// TwinCAT 3 PLC project _710_Clamping
// ProgramVersion: 3.1.4024.0
// libraries:
//   Tc2_Standard, * (Beckhoff Automation GmbH)
//   Tc2_System, * (Beckhoff Automation GmbH)
//   Tc3_Module, * (Beckhoff Automation GmbH)
//   VisuDialogs, * (System)
// project tree:
//   DUTs/ udt_MH_Robot_Input.TcDUT (not stored), udt_HDL_PartData.TcDUT, udt_MH_Robot_Output.TcDUT (not stored)
//   / GlobalTextList.TcGTLO, PlcTask.TcTTO, Visualization Manager.TcVMO (not stored)
//   GVLs/ Inputs.TcGVL (not stored), Memory_DB.TcGVL (not stored), Outputs.TcGVL (not stored)
//   POUs/ Fixture1_Auto.TcPOU, Callblocks.TcPOU, Callblocks_FX1.TcPOU, Callblocks_FX2.TcPOU, Clamp.TcPOU (not stored), Feedback_FB.TcPOU (not stored), Fixture2_Auto.TcPOU (not stored), FX2TextList.TcTLO, MAIN.TcPOU (not stored), MHRobot.TcPOU (not stored), Mode.TcPOU, RollerDoor.TcPOU, FX1TextList.TcTLO, Trunion.TcPOU, Turntable.TcPOU (not stored), WeldRobot.TcPOU (not stored)
//   VISUs/ Fixture_Auto.TcVIS, Fixture_Manual.TcVIS
// real-time tasks:
//   TASK PlcTask: cycle T#10ms, priority 20, ADS port 350

CONFIGURATION _710_Clamping
    RESOURCE PLC ON TwinCAT3
        TASK PlcTask(INTERVAL := T#10ms, PRIORITY := 20);
        PROGRAM MAIN WITH PlcTask : MAIN;
    END_RESOURCE
END_CONFIGURATION

// ---- DUTs/udt_HDL_PartData.TcDUT
TYPE udt_HDL_PartData :
STRUCT
	
PartId	:DINT;
State	:BOOL;
Varient	:BOOL;
Exists	:BOOL;

	
END_STRUCT
END_TYPE

// ---- POUs/Fixture1_Auto.TcPOU
PROGRAM Fixture1_Auto
VAR
	
nState_Door    : INT; // 0: Idle, 10: Starting, 20: Rotating, 30: Stopping
	
END_VAR




/////////////// OPERATOR LOAD PART FIX 1 ///////////////

		IF Memory_DB.M_Auto_Active AND 
		   Memory_DB.M_Power_On AND 
		   Inputs.i_Front_Door_Up
		   THEN   
		IF Memory_DB.M_FX1_LOAD1 AND Memory_DB.M_Turntable_POS1_Reached AND Memory_DB.M_Fixture1_TR_POS1_Reached  THEN
		  Inputs.i_FX1_PART_CONTROL_B1 := TRUE;
		  Inputs.i_FX1_PART_CONTROL_B2 := TRUE;
		  Inputs.i_FX1_PART_CONTROL_B3 := TRUE;
		  Inputs.i_FX1_PART_CONTROL_B4 := TRUE;
		  Inputs.i_FX1_PART_CONTROL_B5 := TRUE;
		  Inputs.i_FX1_PART_CONTROL_B6 := TRUE;
		  Inputs.i_FX1_PART_CONTROL_B7 := TRUE;
		  Memory_DB.M_FX1_LOAD1_COMPLETED :=TRUE;
		
		ELSIF Memory_DB.M_Auto_Active AND Memory_DB.M_Turntable_POS1_Reached AND Memory_DB.M_Fixture1_TR_POS2_Reached AND Memory_DB.M_FX1_LOAD2 THEN
		      Inputs.i_FX1_PART_CONTROL_B15 := TRUE;
		      Inputs.i_FX1_PART_CONTROL_B16 := TRUE;
		      Inputs.i_FX1_PART_CONTROL_B17 := TRUE;
		      Inputs.i_FX1_PART_CONTROL_B18 := TRUE;
		      Inputs.i_FX1_PART_CONTROL_B19 := TRUE;
		      Inputs.i_FX1_PART_CONTROL_B20 := TRUE;
		      Inputs.i_FX1_PART_CONTROL_B21 := TRUE;
		      Memory_DB.M_FX1_LOAD2_COMPLETED :=TRUE;
		
		ELSIF Memory_DB.M_FX1_LOAD1_COMPLETED AND Memory_DB.M_FX1_LOAD2_COMPLETED THEN
			
			  Memory_DB.M_Fixture1_TR_Start :=TRUE;
			
		END_IF;
		END_IF;
		 IF 
		   Memory_DB. M_FX1_All_Initialise THEN
		   Memory_DB.M_Turntable_Start := TRUE;
	       Memory_DB.M_Turntable_POS1_CMD := TRUE;
		   Memory_DB.M_Turntable_POS2_CMD := FALSE;
		   Memory_DB.M_Fixture1_TR_Start := TRUE;
	       Memory_DB.M_Fixture1_TR_POS1_CMD := TRUE;
		   Memory_DB.M_Fixture1_TR_POS2_CMD := FALSE;
		   Memory_DB.M_REAR_DOOR_DOWN := TRUE;
		   Memory_DB.M_REAR_DOOR_Up := FALSE;
		   
		 END_IF
//////////////////LODING SIDE DOOR & TRUNION CONTROL OPERATION/////////////////
IF  Memory_DB.M_Auto_Active AND Memory_DB.M_Safety_Ok AND Memory_DB.M_Power_On  THEN
	
CASE nState_Door  OF
    0: // Default Position1 of Door Open
	IF Memory_DB.M_Turntable_POS1_Reached AND Memory_DB.M_Fixture1_TR_POS1_Reached THEN      
		Memory_DB.M_FRONT_DOOR_Down	:=FALSE;
		Memory_DB.M_FRONT_DOOR_UP	:=TRUE;	
		Memory_DB.M_R03_MH_Goto_Drop2:=FALSE;
		nState_Door := 10;
     END_IF  
	 
    10: // 1st Load completed and Door Close Command
 
        IF Memory_DB.M_FX1_LOAD1_COMPLETED AND Memory_DB.M_FX1_Cycle_Start_PB AND Inputs.i_Front_Door_Up THEN
		Memory_DB.M_FRONT_DOOR_Down	:=TRUE;
		Memory_DB.M_FRONT_DOOR_UP	:=FALSE;

            nState_Door := 20; // Trunion Move
        END_IF
		       
    20: // Clamp Sequence at Trunion Pos1
 
        IF Inputs.i_Front_Door_Down AND Memory_DB.M_Fixture1_TR_POS1_Reached THEN
		Memory_DB.A_FX1_CC1_CLAMPING_UNIT1_3_WP:=TRUE;
		Memory_DB.A_FX1_CC3_CLAMPING_UNIT3_3_WP:=TRUE;
		Memory_DB.A_FX1_CC5_CLAMPING_UNIT5_1_WP:=TRUE;
		Memory_DB.A_FX1_CC1_CLAMPING_UNIT1_3_HP:=FALSE;
		Memory_DB.A_FX1_CC3_CLAMPING_UNIT3_3_HP:=FALSE;
		Memory_DB.A_FX1_CC5_CLAMPING_UNIT5_1_HP:=FALSE;		

         nState_Door := 30; // Error State
        END_IF	

        
    30: // Trunion move to Position 2 for 2nd Load
 
        IF Inputs.i_Front_Door_Down AND Inputs.i_FX1_CC1_Clamp_1_Sensor_WP AND 
		Inputs.i_FX1_CC3_Clamp_1_Sensor_WP AND Inputs.i_FX1_CC5_Clamp_1_Sensor_WP THEN
		Memory_DB.M_Fixture1_TR_POS2_CMD:=TRUE;
		Memory_DB.M_Fixture1_TR_POS1_CMD:=FALSE;

            nState_Door := 40; // Error State
        END_IF		
        
    40: // Door Open command for 2nd Load
 
        IF Memory_DB.M_Fixture1_TR_POS2_Reached AND Inputs.i_Front_Door_Down THEN
		Memory_DB.M_FRONT_DOOR_Down:=FALSE;
		Memory_DB.M_FRONT_DOOR_UP  :=TRUE;

            nState_Door := 50; // Error State
        END_IF	
        
    50: // 2nd Load completed on Trunion & Door Close Command
 
        IF Memory_DB.M_FX1_LOAD2_COMPLETED AND Memory_DB.M_FX1_Cycle_Start_PB AND Inputs.i_Front_Door_Up THEN
		Memory_DB.M_FRONT_DOOR_Down      :=TRUE;
		Memory_DB.M_FRONT_DOOR_Up        :=FALSE;

            nState_Door := 60; // Error State
        END_IF
		
    60: // Clamp Sequence at Trunion Pos1
 
        IF Inputs.i_Front_Door_Down AND Memory_DB.M_Fixture1_TR_POS2_Reached THEN
		Memory_DB.A_FX1_CC2_CLAMPING_UNIT2_3_WP:=TRUE;
		Memory_DB.A_FX1_CC4_CLAMPING_UNIT4_3_WP:=TRUE;
		Memory_DB.A_FX1_CC6_CLAMPING_UNIT6_1_WP:=TRUE;
		Memory_DB.A_FX1_CC2_CLAMPING_UNIT2_3_HP:=FALSE;
		Memory_DB.A_FX1_CC4_CLAMPING_UNIT4_3_HP:=FALSE;
		Memory_DB.A_FX1_CC6_CLAMPING_UNIT6_1_HP:=FALSE;	

         nState_Door := 70; // Error State
        END_IF		
        
    70: // Move Trunion to Default/Pos1
 
        IF Memory_DB.M_Fixture1_TR_Start AND Inputs.i_Front_Door_Down AND Memory_DB.M_Fixture1_TR_POS2_Reached AND
		 Inputs.i_FX1_CC2_Clamp_1_Sensor_WP AND Inputs.i_FX1_CC4_Clamp_1_Sensor_WP AND Inputs.i_FX1_CC6_Clamp_1_Sensor_WP THEN
		Memory_DB.M_Fixture1_TR_POS1_CMD:=TRUE;
		Memory_DB.M_Fixture1_TR_POS2_CMD:=FALSE;

            nState_Door := 80; // Error State
        END_IF
		
    80: // Move TT Work position/Pos2
 
        IF Memory_DB.M_FX1_LOAD1_COMPLETED AND Memory_DB.M_FX1_LOAD2_COMPLETED AND Inputs.i_Front_Door_Down AND Memory_DB.M_Fixture1_TR_POS1_Reached AND Memory_DB.M_Turntable_POS1_Reached 
           AND Inputs.i_Rear_Door_Down AND Inputs.i_FX1_CC2_Clamp_1_Sensor_WP AND Inputs.i_FX1_CC4_Clamp_1_Sensor_WP AND Inputs.i_FX1_CC6_Clamp_1_Sensor_WP 
           AND Memory_DB.M_R01_Home AND Memory_DB.M_R02_Home AND Memory_DB.M_R03_MH_AtHome THEN
		   Memory_DB.M_Turntable_Start:=TRUE;
		   Memory_DB.M_Turntable_POS2_CMD :=TRUE;
		   Memory_DB.M_Turntable_POS1_CMD :=FALSE;
           Memory_DB.M_FRONT_DOOR_Down    :=FALSE;
		   
            nState_Door := 90; // Error State
        END_IF		

	90: // Robot Weld CMD for First Weld
 
       IF  Memory_DB.M_Fixture1_TR_POS1_Reached AND Memory_DB.M_Turntable_POS2_Reached 
           AND Inputs.i_Rear_Door_Down AND Inputs.i_FX1_CC2_Clamp_1_Sensor_WP AND Inputs.i_FX1_CC4_Clamp_1_Sensor_WP AND Inputs.i_FX1_CC6_Clamp_1_Sensor_WP 
           AND Memory_DB.M_R01_Home AND Memory_DB.M_R02_Home AND Memory_DB.M_R03_MH_AtHome THEN
		   Memory_DB.M_R01_Weld_Start:=TRUE;
		   Memory_DB.M_R02_Weld_Start:=TRUE;
		  
            nState_Door := 100; // Error State
      	END_IF			
		
	100: // Trunnion move to POS2 for second Weld
 
        IF Memory_DB.M_R01_Job_Done1 AND Memory_DB.M_R02_Job_Done1 AND Inputs.i_Rear_Door_Down AND Memory_DB.M_Fixture1_TR_POS1_Reached AND Memory_DB.M_Turntable_POS2_Reached AND Inputs.i_FX1_CC2_Clamp_1_Sensor_WP AND Inputs.i_FX1_CC4_Clamp_1_Sensor_WP AND Inputs.i_FX1_CC6_Clamp_1_Sensor_WP THEN
		   Memory_DB.M_Fixture1_TR_POS1_CMD:=FALSE;
		   Memory_DB.M_Fixture1_TR_POS2_CMD:=TRUE;
		  

            nState_Door := 110; // Error State
        END_IF				
		
		
	110: // Robot Weld CMD for Second Weld
 
        IF  Inputs.i_Rear_Door_Down AND Memory_DB.M_Fixture1_TR_POS2_Reached  AND Memory_DB.M_Turntable_POS2_Reached  
           AND Inputs.i_FX1_CC2_Clamp_1_Sensor_WP AND Inputs.i_FX1_CC4_Clamp_1_Sensor_WP AND Inputs.i_FX1_CC6_Clamp_1_Sensor_WP THEN
		   Memory_DB.M_R01_Weld_Start:=TRUE;
		   Memory_DB.M_R02_Weld_Start:=TRUE;
		  
            nState_Door := 120; // Error State
        END_IF					
		
		
	120: // Trunnion move to POS1 for Unload part
 
        IF Memory_DB.M_R01_Job_Done1 AND Memory_DB.M_R02_Job_Done1 AND Memory_DB.M_R01_Job_Done2 AND Memory_DB.M_R02_Job_Done2 AND Inputs.i_Rear_Door_Down AND Memory_DB.M_Fixture1_TR_POS2_Reached AND Memory_DB.M_Turntable_POS2_Reached AND Inputs.i_FX1_CC2_Clamp_1_Sensor_WP AND Inputs.i_FX1_CC4_Clamp_1_Sensor_WP AND Inputs.i_FX1_CC6_Clamp_1_Sensor_WP THEN
		   Memory_DB.M_Fixture1_TR_POS2_CMD :=FALSE;
		   Memory_DB.M_Fixture1_TR_POS1_CMD :=TRUE;
		   Memory_DB.M_R01_Weld_Start:=FALSE;
		   Memory_DB.M_R02_Weld_Start:=FALSE;
		   
            nState_Door := 130; // Error State
        END_IF					
		
			
	130: // Rear Door Open
 
        IF  Inputs.i_Rear_Door_Down AND Memory_DB.M_Fixture1_TR_POS1_Reached AND Memory_DB.M_Turntable_POS2_Reached AND Inputs.i_FX1_CC2_Clamp_1_Sensor_WP AND Inputs.i_FX1_CC4_Clamp_1_Sensor_WP AND Inputs.i_FX1_CC6_Clamp_1_Sensor_WP THEN
		   Memory_DB.M_Rear_DOOR_Up      :=TRUE;
		   Memory_DB.M_Rear_DOOR_Down    :=FALSE;
		  
		   
            nState_Door := 140; // Error State
        END_IF
	
		
	140: // MH Robot Part Unload Command
 
        IF Inputs.i_Rear_Door_Up AND Memory_DB.M_Fixture1_TR_POS1_Reached AND Memory_DB.M_Turntable_POS2_Reached AND Inputs.i_FX1_CC2_Clamp_1_Sensor_WP AND Inputs.i_FX1_CC4_Clamp_1_Sensor_WP AND Inputs.i_FX1_CC6_Clamp_1_Sensor_WP THEN
		   Memory_DB.M_R03_MH_Cycle_Start   :=TRUE;
		   Memory_DB.M_R03_MH_MovePounce    :=TRUE;
		  
		   
            nState_Door := 150; // Error State
        END_IF
	
	150: // MH Robot At Pounce and Fixture Clamp Open
 
     IF Memory_DB.M_R03_MH_MovePounce AND Inputs.i_Rear_Door_Up AND Memory_DB.M_Fixture1_TR_POS1_Reached AND Memory_DB.M_Turntable_POS2_Reached AND Inputs.i_FX1_CC1_Clamp_1_Sensor_WP AND Inputs.i_FX1_CC3_Clamp_1_Sensor_WP AND Inputs.i_FX1_CC5_Clamp_1_Sensor_WP THEN
		Memory_DB.A_FX1_CC1_CLAMPING_UNIT1_3_HP:=TRUE;
		Memory_DB.A_FX1_CC3_CLAMPING_UNIT3_3_HP:=TRUE;
		Memory_DB.A_FX1_CC5_CLAMPING_UNIT5_1_HP:=TRUE;
		Memory_DB.A_FX1_CC1_CLAMPING_UNIT1_3_WP:=FALSE;
		Memory_DB.A_FX1_CC3_CLAMPING_UNIT3_3_WP:=FALSE;
		Memory_DB.A_FX1_CC5_CLAMPING_UNIT5_1_WP:=FALSE;	
		  
		   
            nState_Door := 160; // Error State
     END_IF
	 
	 
	160: // MH Robot Part Pick1 Command
 
        IF Inputs.i_Rear_Door_Up AND Memory_DB.M_Fixture1_TR_POS1_Reached AND Memory_DB.M_Turntable_POS2_Reached AND Inputs.i_FX1_CC1_Clamp_1_Sensor_HP AND Inputs.i_FX1_CC3_Clamp_1_Sensor_HP AND Inputs.i_FX1_CC5_Clamp_1_Sensor_HP THEN
		   Memory_DB.M_R03_MH_Cycle_Start   :=FALSE;
		   Memory_DB.M_R03_MH_MovePounce    :=FALSE;
		  Memory_DB.M_R03_MH_Goto_Pick1     :=TRUE;
		  Inputs.i_FX1_PART_CONTROL_B1 := FALSE;
		  Inputs.i_FX1_PART_CONTROL_B2 := FALSE;
		  Inputs.i_FX1_PART_CONTROL_B3 := FALSE;
		  Inputs.i_FX1_PART_CONTROL_B4 := FALSE;
		  Inputs.i_FX1_PART_CONTROL_B5 := FALSE;
		  Inputs.i_FX1_PART_CONTROL_B6 := FALSE;
		  Inputs.i_FX1_PART_CONTROL_B7 := FALSE;
		   
            nState_Door := 170; // Error State
        END_IF	
		
		
	170: // MH Robot Move to Paunce 
 
        IF Inputs.i_Rear_Door_Up AND Memory_DB.M_Fixture1_TR_POS1_Reached AND Memory_DB.M_Turntable_POS2_Reached AND Inputs.i_FX1_CC2_Clamp_1_Sensor_WP AND Inputs.i_FX1_CC4_Clamp_1_Sensor_WP AND Inputs.i_FX1_CC6_Clamp_1_Sensor_WP THEN
		  
		   Memory_DB.M_R03_MH_MovePounce    :=TRUE;	  
		   
            nState_Door := 180; // Error State
        END_IF		
		
	180: // Trunion rotate to Pos2
 
        IF Inputs.i_Rear_Door_Up AND Memory_DB.M_R03_MH_Pick1_Done AND Memory_DB.M_Fixture1_TR_POS1_Reached AND Memory_DB.M_Turntable_POS2_Reached AND Inputs.i_FX1_CC2_Clamp_1_Sensor_WP AND Inputs.i_FX1_CC4_Clamp_1_Sensor_WP AND Inputs.i_FX1_CC6_Clamp_1_Sensor_WP THEN
		   Memory_DB.M_Fixture1_TR_POS1_CMD:=FALSE;
		   Memory_DB.M_Fixture1_TR_POS2_CMD:=TRUE;
		    		   
            nState_Door := 190; // Error State
        END_IF		
			
	190: // Fixture clamp Open
 
       IF Inputs.i_Rear_Door_Up AND Memory_DB.M_R03_MH_Pick1_Done AND Memory_DB.M_Fixture1_TR_POS2_Reached AND Memory_DB.M_Turntable_POS2_Reached AND Inputs.i_FX1_CC2_Clamp_1_Sensor_WP AND Inputs.i_FX1_CC4_Clamp_1_Sensor_WP AND Inputs.i_FX1_CC6_Clamp_1_Sensor_WP THEN
		Memory_DB.A_FX1_CC2_CLAMPING_UNIT2_3_HP:=TRUE;
		Memory_DB.A_FX1_CC4_CLAMPING_UNIT4_3_HP:=TRUE;
		Memory_DB.A_FX1_CC6_CLAMPING_UNIT6_1_HP:=TRUE;
		Memory_DB.A_FX1_CC2_CLAMPING_UNIT2_3_WP:=FALSE;
		Memory_DB.A_FX1_CC4_CLAMPING_UNIT4_3_WP:=FALSE;
		Memory_DB.A_FX1_CC6_CLAMPING_UNIT6_1_WP:=FALSE;	
		    		   
            nState_Door := 200; // Error State
       END_IF			
		
	  200: // MH Robot Part Pick2 Command
 
       IF Inputs.i_Rear_Door_Up AND Memory_DB.M_R03_MH_Pick1_Done AND Memory_DB.M_Fixture1_TR_POS2_Reached AND Memory_DB.M_Turntable_POS2_Reached AND Inputs.i_FX1_CC2_Clamp_1_Sensor_HP AND Inputs.i_FX1_CC4_Clamp_1_Sensor_HP AND Inputs.i_FX1_CC6_Clamp_1_Sensor_HP THEN
		  Memory_DB.M_R03_MH_MovePounce    :=FALSE;
		  Memory_DB.M_R03_MH_Goto_Pick2     :=TRUE;
		  Inputs.i_FX1_PART_CONTROL_B15 := FALSE;
		  Inputs.i_FX1_PART_CONTROL_B16 := FALSE;
		  Inputs.i_FX1_PART_CONTROL_B17 := FALSE;
		  Inputs.i_FX1_PART_CONTROL_B18 := FALSE;
		  Inputs.i_FX1_PART_CONTROL_B19 := FALSE;
		  Inputs.i_FX1_PART_CONTROL_B20 := FALSE;
		  Inputs.i_FX1_PART_CONTROL_B21 := FALSE;
		    		   
            nState_Door := 210; // Error State
       END_IF	
 
	 210: // Trunion rotate to POS1  
	   IF Inputs.i_Rear_Door_Up AND Memory_DB.M_R03_MH_Pick1_Done AND Memory_DB.M_Fixture1_TR_POS2_Reached AND Memory_DB.M_Turntable_POS2_Reached AND Inputs.i_FX1_CC2_Clamp_1_Sensor_HP AND Inputs.i_FX1_CC4_Clamp_1_Sensor_HP AND Inputs.i_FX1_CC6_Clamp_1_Sensor_HP THEN
		  Memory_DB.M_Fixture1_TR_POS1_CMD := TRUE;
		  Memory_DB.M_Fixture1_TR_POS2_CMD := FALSE; 
		  
		    		   
            nState_Door := 220; // Error State
       END_IF	 
	   
	 220: // Rear Door Down
 
       IF Inputs.i_Rear_Door_Up AND Memory_DB.M_R03_MH_Pick1_Done AND Memory_DB.M_R03_MH_Pick2_Done AND Memory_DB.M_Fixture1_TR_POS1_Reached AND Memory_DB.M_Turntable_POS2_Reached THEN
		   Memory_DB.M_Rear_DOOR_Down   :=TRUE;
		   Memory_DB.M_Rear_DOOR_Up     :=FALSE;
		  Memory_DB.M_R03_MH_MovePounce :=TRUE;
		  Memory_DB.M_R01_Job_Done1     :=FALSE;   
		  Memory_DB.M_R01_Job_Done2     :=FALSE;    
          Memory_DB.M_R02_Job_Done1     :=FALSE;  
		  Memory_DB.M_R02_Job_Done2     :=FALSE;   
          Memory_DB.M_R03_MH_Goto_Pick1 :=FALSE; 
		  Memory_DB.M_R03_MH_Goto_Pick2 :=FALSE;
            nState_Door := 230; // Error State
       END_IF	
 	
	
	    230: // Robot Go to Drop1 & Drop2
 
       IF Inputs.i_Rear_Door_Down AND Memory_DB.M_R03_MH_Pick1_Done AND Memory_DB.M_R03_MH_Pick2_Done AND Memory_DB.M_Fixture1_TR_POS1_Reached AND Memory_DB.M_Turntable_POS2_Reached THEN
		  
		  Memory_DB.M_R03_MH_Goto_Drop1 :=TRUE;	    
		  Memory_DB.M_R03_MH_MovePounce :=FALSE;  
		   
 
            nState_Door := 240; // Error State
       END_IF
	
	   240: // Robot Go to Drop2 
 
       IF Inputs.i_Rear_Door_Down AND Memory_DB.M_R03_MH_Pick1_Done AND Memory_DB.M_R03_MH_Pick2_Done AND Memory_DB.M_Fixture1_TR_POS1_Reached AND Memory_DB.M_Turntable_POS2_Reached THEN
		  
		  Memory_DB.M_R03_MH_Goto_Drop1 :=FALSE;
		  Memory_DB.M_R03_MH_Goto_Drop2  :=TRUE;   
		  Memory_DB.M_R03_MH_MovePounce :=FALSE;  
		  
 
            nState_Door := 250; // Error State
       END_IF

	 250: // TT Rotate to load position 
 
       IF Memory_DB.M_Fixture1_TR_POS1_Reached AND Memory_DB.M_Turntable_POS1_Reached THEN
		  	   
 
            nState_Door := 0; // Error State
       END_IF
END_CASE;
END_IF;

END_PROGRAM

// ---- POUs/Callblocks.TcPOU
PROGRAM Callblocks
VAR
	
Temp_bool : BOOL;
Mode_0          : Mode;
Feedback_FD     : Feedback_FB;
Feedback_RD     : Feedback_FB;
Feedback_FX1TR  : Feedback_FB;
Feedback_FX2TR  : Feedback_FB;
Feedback_TT     : Feedback_FB;
Feedback_CL     : Feedback_FB;

Front_Door        : RollerDoor;
Rear_Door         : RollerDoor;
Fixture1_Trunion  : Trunion;
Fixture2_Trunion  : Trunion;
TT                : Turntable ;
Robot1            : Weldrobot;
Robot2            : Weldrobot;



	
	MHRobot_0: MHRobot;
END_VAR

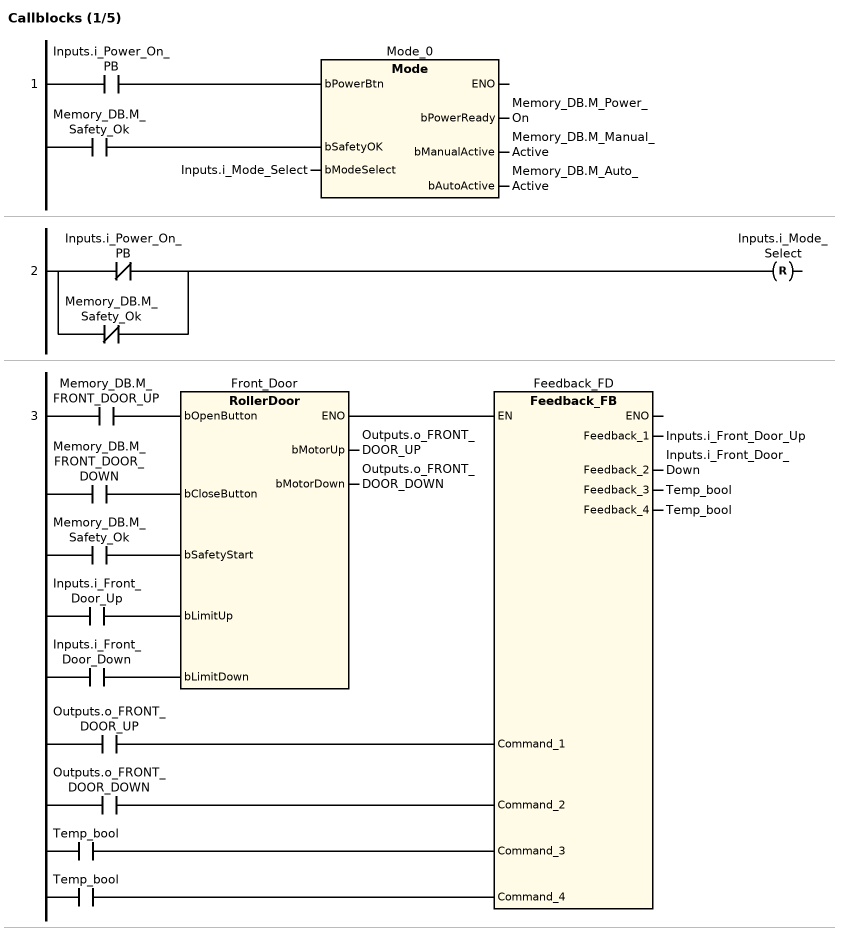
// NETWORK 1
Mode_0(
    bPowerBtn := Inputs.i_Power_On_PB,
    bSafetyOK := Memory_DB.M_Safety_Ok,
    bModeSelect := Inputs.i_Mode_Select,
    bPowerReady => Memory_DB.M_Power_On,
    bManualActive => Memory_DB.M_Manual_Active,
    bAutoActive => Memory_DB.M_Auto_Active); // Mode

// NETWORK 2
Inputs.i_Mode_Select R= NOT Inputs.i_Power_On_PB OR NOT Memory_DB.M_Safety_Ok;

// NETWORK 3
Front_Door(
    bOpenButton := Memory_DB.M_FRONT_DOOR_UP,
    bCloseButton := Memory_DB.M_FRONT_DOOR_DOWN,
    bSafetyStart := Memory_DB.M_Safety_Ok,
    bLimitUp := Inputs.i_Front_Door_Up,
    bLimitDown := Inputs.i_Front_Door_Down,
    bMotorUp => Outputs.o_FRONT_DOOR_UP,
    bMotorDown => Outputs.o_FRONT_DOOR_DOWN); // RollerDoor
Feedback_FD(
    EN := TRUE,
    Command_1 := Outputs.o_FRONT_DOOR_UP,
    Command_2 := Outputs.o_FRONT_DOOR_DOWN,
    Command_3 := Temp_bool,
    Command_4 := Temp_bool,
    Feedback_1 => Inputs.i_Front_Door_Up,
    Feedback_2 => Inputs.i_Front_Door_Down,
    Feedback_3 => Temp_bool,
    Feedback_4 => Temp_bool); // Feedback_FB

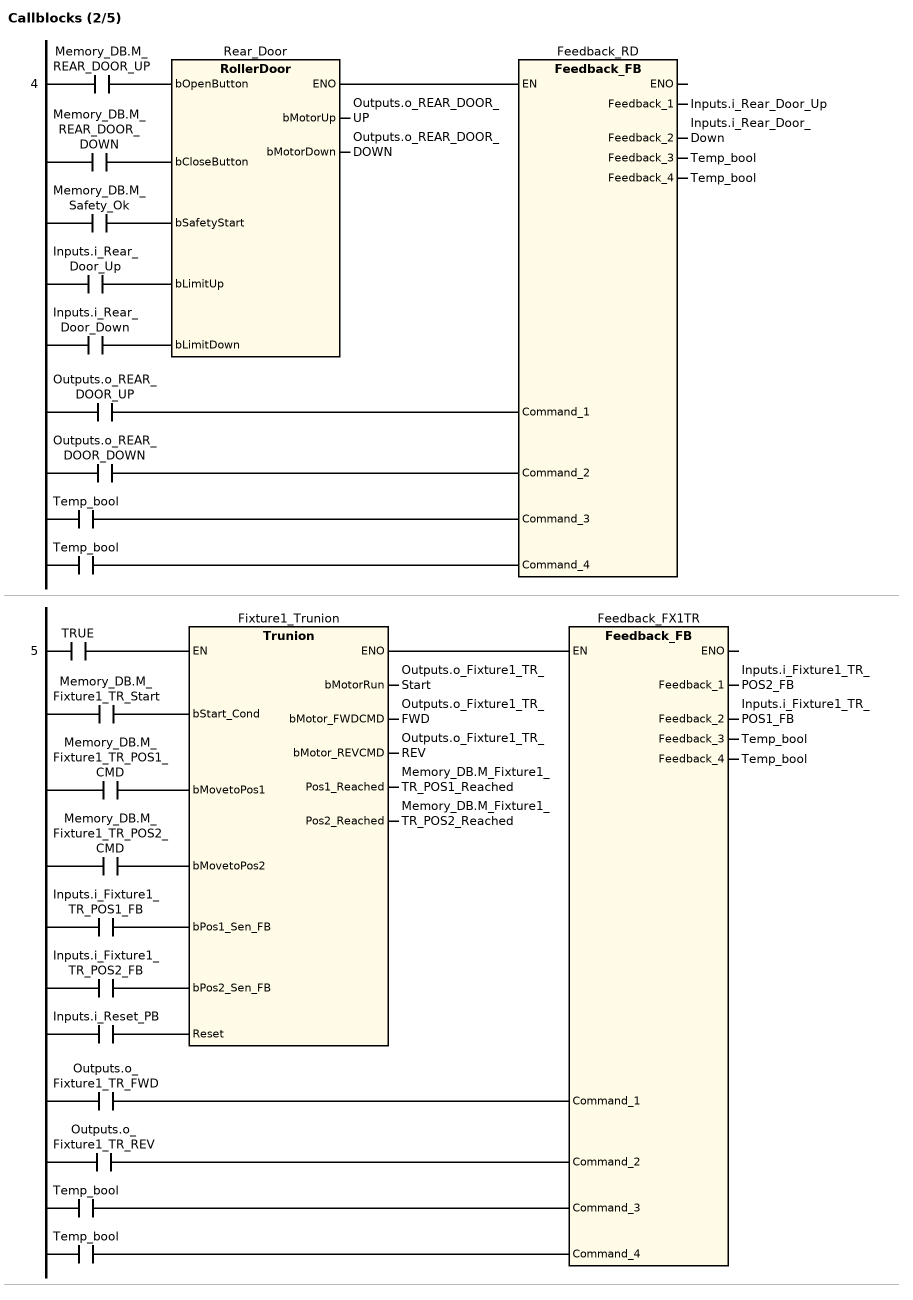
// NETWORK 4
Rear_Door(
    bOpenButton := Memory_DB.M_REAR_DOOR_UP,
    bCloseButton := Memory_DB.M_REAR_DOOR_DOWN,
    bSafetyStart := Memory_DB.M_Safety_Ok,
    bLimitUp := Inputs.i_Rear_Door_Up,
    bLimitDown := Inputs.i_Rear_Door_Down,
    bMotorUp => Outputs.o_REAR_DOOR_UP,
    bMotorDown => Outputs.o_REAR_DOOR_DOWN); // RollerDoor
Feedback_RD(
    EN := TRUE,
    Command_1 := Outputs.o_REAR_DOOR_UP,
    Command_2 := Outputs.o_REAR_DOOR_DOWN,
    Command_3 := Temp_bool,
    Command_4 := Temp_bool,
    Feedback_1 => Inputs.i_Rear_Door_Up,
    Feedback_2 => Inputs.i_Rear_Door_Down,
    Feedback_3 => Temp_bool,
    Feedback_4 => Temp_bool); // Feedback_FB

// NETWORK 5
Fixture1_Trunion(
    EN := TRUE,
    bStart_Cond := Memory_DB.M_Fixture1_TR_Start,
    bMovetoPos1 := Memory_DB.M_Fixture1_TR_POS1_CMD,
    bMovetoPos2 := Memory_DB.M_Fixture1_TR_POS2_CMD,
    bPos1_Sen_FB := Inputs.i_Fixture1_TR_POS1_FB,
    bPos2_Sen_FB := Inputs.i_Fixture1_TR_POS2_FB,
    Reset := Inputs.i_Reset_PB,
    bMotorRun => Outputs.o_Fixture1_TR_Start,
    bMotor_FWDCMD => Outputs.o_Fixture1_TR_FWD,
    bMotor_REVCMD => Outputs.o_Fixture1_TR_REV,
    Pos1_Reached => Memory_DB.M_Fixture1_TR_POS1_Reached,
    Pos2_Reached => Memory_DB.M_Fixture1_TR_POS2_Reached); // Trunion
Feedback_FX1TR(
    EN := TRUE,
    Command_1 := Outputs.o_Fixture1_TR_FWD,
    Command_2 := Outputs.o_Fixture1_TR_REV,
    Command_3 := Temp_bool,
    Command_4 := Temp_bool,
    Feedback_1 => Inputs.i_Fixture1_TR_POS2_FB,
    Feedback_2 => Inputs.i_Fixture1_TR_POS1_FB,
    Feedback_3 => Temp_bool,
    Feedback_4 => Temp_bool); // Feedback_FB

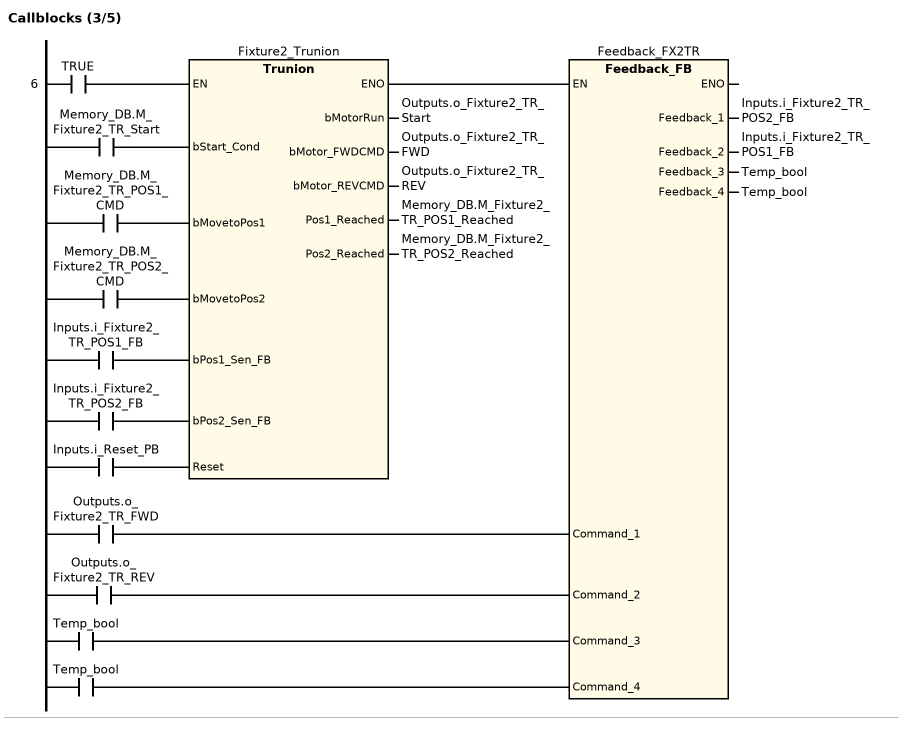
// NETWORK 6
Fixture2_Trunion(
    EN := TRUE,
    bStart_Cond := Memory_DB.M_Fixture2_TR_Start,
    bMovetoPos1 := Memory_DB.M_Fixture2_TR_POS1_CMD,
    bMovetoPos2 := Memory_DB.M_Fixture2_TR_POS2_CMD,
    bPos1_Sen_FB := Inputs.i_Fixture2_TR_POS1_FB,
    bPos2_Sen_FB := Inputs.i_Fixture2_TR_POS2_FB,
    Reset := Inputs.i_Reset_PB,
    bMotorRun => Outputs.o_Fixture2_TR_Start,
    bMotor_FWDCMD => Outputs.o_Fixture2_TR_FWD,
    bMotor_REVCMD => Outputs.o_Fixture2_TR_REV,
    Pos1_Reached => Memory_DB.M_Fixture2_TR_POS1_Reached,
    Pos2_Reached => Memory_DB.M_Fixture2_TR_POS2_Reached); // Trunion
Feedback_FX2TR(
    EN := TRUE,
    Command_1 := Outputs.o_Fixture2_TR_FWD,
    Command_2 := Outputs.o_Fixture2_TR_REV,
    Command_3 := Temp_bool,
    Command_4 := Temp_bool,
    Feedback_1 => Inputs.i_Fixture2_TR_POS2_FB,
    Feedback_2 => Inputs.i_Fixture2_TR_POS1_FB,
    Feedback_3 => Temp_bool,
    Feedback_4 => Temp_bool); // Feedback_FB

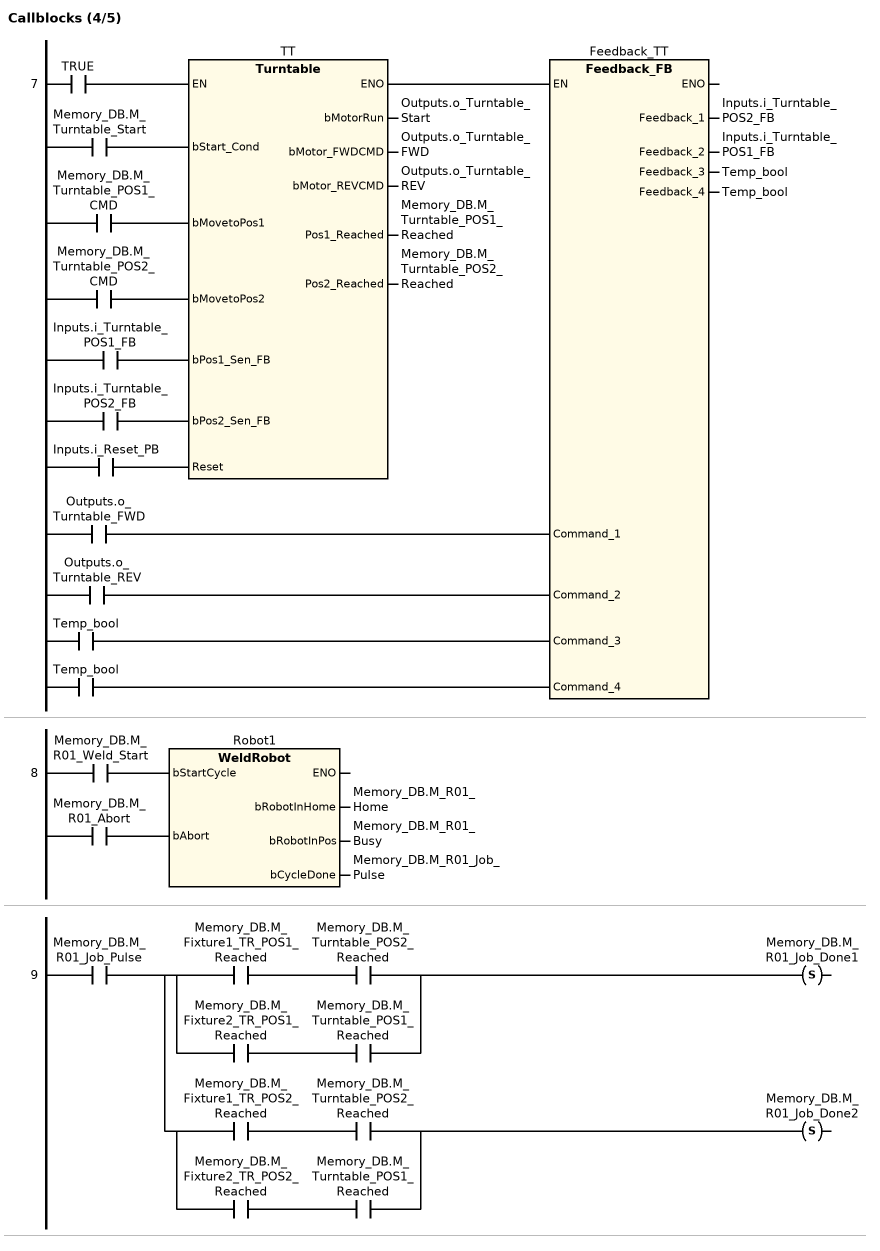
// NETWORK 7
TT(
    EN := TRUE,
    bStart_Cond := Memory_DB.M_Turntable_Start,
    bMovetoPos1 := Memory_DB.M_Turntable_POS1_CMD,
    bMovetoPos2 := Memory_DB.M_Turntable_POS2_CMD,
    bPos1_Sen_FB := Inputs.i_Turntable_POS1_FB,
    bPos2_Sen_FB := Inputs.i_Turntable_POS2_FB,
    Reset := Inputs.i_Reset_PB,
    bMotorRun => Outputs.o_Turntable_Start,
    bMotor_FWDCMD => Outputs.o_Turntable_FWD,
    bMotor_REVCMD => Outputs.o_Turntable_REV,
    Pos1_Reached => Memory_DB.M_Turntable_POS1_Reached,
    Pos2_Reached => Memory_DB.M_Turntable_POS2_Reached); // Turntable
Feedback_TT(
    EN := TRUE,
    Command_1 := Outputs.o_Turntable_FWD,
    Command_2 := Outputs.o_Turntable_REV,
    Command_3 := Temp_bool,
    Command_4 := Temp_bool,
    Feedback_1 => Inputs.i_Turntable_POS2_FB,
    Feedback_2 => Inputs.i_Turntable_POS1_FB,
    Feedback_3 => Temp_bool,
    Feedback_4 => Temp_bool); // Feedback_FB

// NETWORK 8
Robot1(
    bStartCycle := Memory_DB.M_R01_Weld_Start,
    bAbort := Memory_DB.M_R01_Abort,
    bRobotInHome => Memory_DB.M_R01_Home,
    bRobotInPos => Memory_DB.M_R01_Busy,
    bCycleDone => Memory_DB.M_R01_Job_Pulse); // WeldRobot

// NETWORK 9
Memory_DB.M_R01_Job_Done1 S= (Memory_DB.M_R01_Job_Pulse AND Memory_DB.M_Fixture1_TR_POS1_Reached) AND Memory_DB.M_Turntable_POS2_Reached OR (Memory_DB.M_R01_Job_Pulse AND Memory_DB.M_Fixture2_TR_POS1_Reached) AND Memory_DB.M_Turntable_POS1_Reached;
Memory_DB.M_R01_Job_Done2 S= (Memory_DB.M_R01_Job_Pulse AND Memory_DB.M_Fixture1_TR_POS2_Reached) AND Memory_DB.M_Turntable_POS2_Reached OR (Memory_DB.M_R01_Job_Pulse AND Memory_DB.M_Fixture2_TR_POS2_Reached) AND Memory_DB.M_Turntable_POS1_Reached;

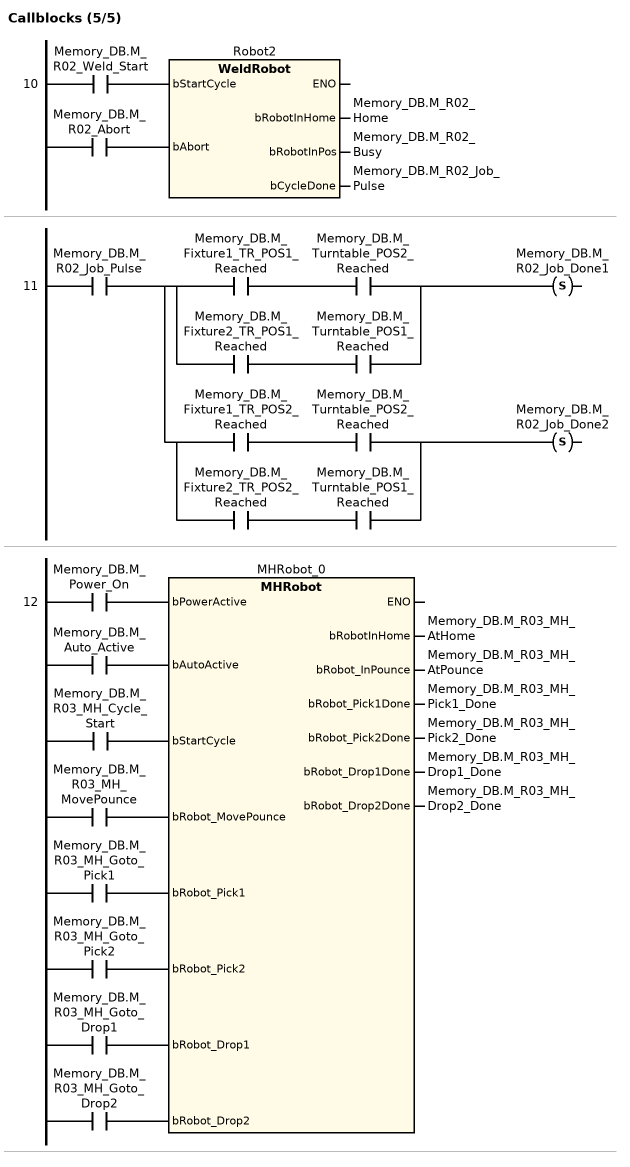
// NETWORK 10
Robot2(
    bStartCycle := Memory_DB.M_R02_Weld_Start,
    bAbort := Memory_DB.M_R02_Abort,
    bRobotInHome => Memory_DB.M_R02_Home,
    bRobotInPos => Memory_DB.M_R02_Busy,
    bCycleDone => Memory_DB.M_R02_Job_Pulse); // WeldRobot

// NETWORK 11
Memory_DB.M_R02_Job_Done1 S= (Memory_DB.M_R02_Job_Pulse AND Memory_DB.M_Fixture1_TR_POS1_Reached) AND Memory_DB.M_Turntable_POS2_Reached OR (Memory_DB.M_R02_Job_Pulse AND Memory_DB.M_Fixture2_TR_POS1_Reached) AND Memory_DB.M_Turntable_POS1_Reached;
Memory_DB.M_R02_Job_Done2 S= (Memory_DB.M_R02_Job_Pulse AND Memory_DB.M_Fixture1_TR_POS2_Reached) AND Memory_DB.M_Turntable_POS2_Reached OR (Memory_DB.M_R02_Job_Pulse AND Memory_DB.M_Fixture2_TR_POS2_Reached) AND Memory_DB.M_Turntable_POS1_Reached;

// NETWORK 12
MHRobot_0(
    bPowerActive := Memory_DB.M_Power_On,
    bAutoActive := Memory_DB.M_Auto_Active,
    bStartCycle := Memory_DB.M_R03_MH_Cycle_Start,
    bRobot_MovePounce := Memory_DB.M_R03_MH_MovePounce,
    bRobot_Pick1 := Memory_DB.M_R03_MH_Goto_Pick1,
    bRobot_Pick2 := Memory_DB.M_R03_MH_Goto_Pick2,
    bRobot_Drop1 := Memory_DB.M_R03_MH_Goto_Drop1,
    bRobot_Drop2 := Memory_DB.M_R03_MH_Goto_Drop2,
    bRobotInHome => Memory_DB.M_R03_MH_AtHome,
    bRobot_InPounce => Memory_DB.M_R03_MH_AtPounce,
    bRobot_Pick1Done => Memory_DB.M_R03_MH_Pick1_Done,
    bRobot_Pick2Done => Memory_DB.M_R03_MH_Pick2_Done,
    bRobot_Drop1Done => Memory_DB.M_R03_MH_Drop1_Done,
    bRobot_Drop2Done => Memory_DB.M_R03_MH_Drop2_Done); // MHRobot

END_PROGRAM

// ---- POUs/Mode.TcPOU
FUNCTION_BLOCK PUBLIC Mode
VAR_INPUT
	 // --- Inputs (HMI or Physical) ---
    bPowerBtn       : BOOL;    // Main Power Toggle
    bSafetyOK       : BOOL;    // Global Safety Signal
    
    bModeSelect     : BOOL;
END_VAR
VAR_OUTPUT
	
	// --- Outputs (Physical or HMI Status) ---
	ENO             : BOOL;
	bPowerReady     : BOOL;    // Power stage is energized
    bManualActive   : BOOL;    // Manual mode is live
    bAutoActive     : BOOL;    // Auto sequence is live
    
	
	
END_VAR
VAR
 // --- Internal Status ---
    bSystemError    : BOOL;    // Power-up failure or safety trip
    nStatePower     : INT;     // State machine for power-up	
	 // --- Timers ---
    tPowerTimer     : TON;     // Simulation for contactors
	nModeSelect     : INT;     // 0:Off, 1:Manual, 2:Auto
END_VAR

// 1. SAFETY INTERLOCK
// If safety trips, everything stops immediately

IF bModeSelect THEN
	nModeSelect :=1;
ELSE
	nModeSelect :=0;	
	
END_IF
IF NOT bSafetyOK THEN
    bPowerReady   := FALSE;
    bManualActive := FALSE;
    bAutoActive   := FALSE;
    nStatePower   := 0;
    bSystemError  := TRUE;
END_IF

// 2. POWER ON STATE MACHINE
CASE nStatePower OF
    0: // IDLE: Waiting for Power Button
        IF bPowerBtn AND bSafetyOK THEN
            nStatePower := 10;
        END_IF
        
    10: // ENERGIZING: Waiting for hardware feedback
        tPowerTimer(IN := TRUE, PT := T#1.5S);
        IF tPowerTimer.Q THEN
            tPowerTimer(IN := FALSE);
            bPowerReady := TRUE;
            bSystemError := FALSE;
            nStatePower := 20;
        END_IF
        
    20: // POWER READY: Monitoring
        IF NOT bPowerBtn OR NOT bSafetyOK THEN
            bPowerReady := FALSE;
            nStatePower := 0;
        END_IF
END_CASE

// 3. MODE SELECTION & OUTPUTS
// Active outputs are ONLY possible if bPowerReady is TRUE
IF bPowerReady THEN
    
    // Mode Logic
    CASE nModeSelect OF
        0: // Manual Selected
            bManualActive := TRUE;
            bAutoActive   := FALSE;
            
        1: // Auto Selected
            bManualActive := FALSE;
            bAutoActive   := TRUE;
            
        ELSE // Off or Invalid
            bManualActive := FALSE;
            bAutoActive   := FALSE;
    END_CASE
    
ELSE
    // Force all active outputs OFF if power is lost
    bManualActive := FALSE;
    bAutoActive   := FALSE;
END_IF

END_FUNCTION_BLOCK

// ---- POUs/RollerDoor.TcPOU
FUNCTION_BLOCK PUBLIC RollerDoor
VAR_INPUT
	
    bOpenButton     : BOOL;     // Pushbutton / Pull-cord
    bCloseButton    : BOOL;     // Pushbutton
    bSafetyStart     : BOOL;     // Bottom edge sensor (Normally Closed for safety)
    bLimitUp        : BOOL;     // Door fully open sensor
    bLimitDown      : BOOL;     // Door fully closed sensor


END_VAR
VAR_OUTPUT
	ENO             : BOOL;
    bMotorUp        : BOOL;     // Up Contactor
    bMotorDown      : BOOL;     // Down Contactor

END_VAR
VAR
	
    nState          : INT;      // 0: Stopped, 10: Opening, 20: Closing, 99: Error
    fbAutoCloseTimer: TON;      // Automatically close after opening

END_VAR

// Auto-Close Timer: Starts when door is fully open
fbAutoCloseTimer(IN := bLimitUp, PT := T#10S);

CASE nState OF
    0: // STOPPED
       // bMotorUp   := FALSE;
       // bMotorDown := FALSE;
        
        IF bOpenButton AND bSafetyStart AND NOT bCloseButton AND NOT bLimitUp THEN
            nState := 10;
        ELSIF bCloseButton AND bSafetyStart AND NOT bOpenButton AND NOT bLimitDown THEN
            // Only allow closing if safety is clear
         
                nState := 20;
           
        END_IF

    10: // OPENING
        bMotorUp   := TRUE;
        bMotorDown := FALSE;
        
        IF bLimitUp THEN
           nState := 0; // Stop if reached limit or close pressed
        END_IF

    20: // CLOSING
        bMotorUp   := FALSE;
        bMotorDown := TRUE;
        
        // Safety Reversal: If something is hit or detected, open immediately
       IF bLimitdown  THEN
           nState := 0;
       END_IF

    99: // ERROR / EMERGENCY STOP
        bMotorUp   := FALSE;
        bMotorDown := FALSE;
END_CASE

END_FUNCTION_BLOCK

// ---- POUs/Trunion.TcPOU
FUNCTION_BLOCK PUBLIC Trunion
VAR_INPUT
	EN : BOOL;
	bStart_Cond     : BOOL;     // Start rotation command
	bMovetoPos1 	: BOOL;   // Move to position 1 / default postion
	bMovetoPos2 	: BOOL;   // Move to position 1
    bPos1_Sen_FB    : BOOL;     // Proximity sensor for position 
    bPos2_Sen_FB    : BOOL;     // Proximity sensor for position  
  	Reset		    : BOOL;
END_VAR

VAR_OUTPUT
 ENO 			: BOOL;	
 bMotorRun   	: BOOL;     // Command to the motor/drive
 bMotor_FWDCMD  : BOOL;     // Motor Forward Command
 bMotor_REVCMD  : BOOL;     // Motor Reverse Command
Pos1_Reached 	: BOOL;   // Default position reached memory
Pos2_Reached	:BOOL;   // 2nd position reached memory
	

END_VAR

VAR	
    nState          : INT; // 0: Idle, 10: Starting, 20: Rotating, 30: Stopping
    fbTimeout       : TON;      // Safety timeout timer
	sAlarm          : STRING;   // Error message

END_VAR

CASE nState OF
    0: // IDLE - Default Position1
	 
		IF bMovetoPos2 AND NOT bMovetoPos1 THEN
			nState := 10;
		ELSIF bMovetoPos1 AND NOT bMovetoPos2 THEN
			nState := 30;
		END_IF;

        
    10: // Move to 2nd position
        bMotor_REVCMD  := FALSE;
        bMotor_FWDCMD := TRUE;
        
        IF Pos2_Reached THEN
            nState := 0;
			bMotor_FWDCMD := FALSE;
        ELSIF fbTimeout.Q THEN
            sAlarm := 'Error: Pos2 Timeout';
            nState := 99; // Error State
        END_IF
        
        
    30: // Move to 1st position
        bMotor_FWDCMD := FALSE;
        bMotor_revCMD  := TRUE;
        
        IF Pos1_Reached THEN
            nState := 0;
			bMotor_REVCMD := FALSE;
        ELSIF fbTimeout.Q THEN
            sAlarm := 'Error: Pos1 Timeout';
            nState := 99;
        END_IF
		
	99: // ERROR STATE
        bMotor_FWDCMD := FALSE;
        bMotor_revCMD  := FALSE; // De-energize for safety
        IF NOT bMovetoPos2 AND NOT bMovetoPos1 THEN
            nState := 0; // Reset after clearing request
        END_IF

 END_CASE


IF NOT bStart_Cond  THEN
	    bMotor_FWDCMD := FALSE;
        bMotor_revCMD  := FALSE;
END_IF;

/////// ERROR ACKNOWLEDGE/////////////////

IF reset THEN
	sAlarm := '';
	
	END_IF;

////MOTOR RUN COMMANE OUTPUT/////////////
IF bMotor_FWDCMD OR bMotor_REVCMD THEN
	bMotorRun:= TRUE;
	ELSE 
		bMotorRun:= FALSE;
	END_IF

/// POSITION REACHED MEMORY FIRE ////////
IF bPos1_Sen_FB AND bMotor_REVCMD THEN
Pos1_Reached:= TRUE;
ELSIF bMotor_fwdCMD THEN
Pos1_Reached:= FALSE;
END_IF;

/// POSITION REACHED MEMORY FIRE ////////
IF bPos2_Sen_FB AND bMotor_fwdCMD THEN
Pos2_Reached:= TRUE;
ELSIF bMotor_revCMD THEN
Pos2_Reached:= FALSE;
END_IF;

END_FUNCTION_BLOCK

// ---- POUs/Callblocks_FX1.TcPOU
PROGRAM Callblocks_FX1
VAR
	
FX1_CC1_Clamp_Unit1_3 : clamp;
FX1_CC2_Clamp_Unit2_3 : clamp;
FX1_CC3_Clamp_Unit3_3 : clamp;
FX1_CC4_Clamp_Unit4_3 : clamp;
FX1_CC5_Clamp_Unit5_1 : clamp;
FX1_CC6_Clamp_Unit6_1 : clamp;

Temp_bool : BOOL;
FX1_Feedback_Unit1  : Feedback_FB;
FX1_Feedback_Unit2  : Feedback_FB;
FX1_Feedback_Unit3  : Feedback_FB;
FX1_Feedback_Unit4  : Feedback_FB;
FX1_Feedback_Unit5  : Feedback_FB;
FX1_Feedback_Unit6  : Feedback_FB;


END_VAR
VAR // added by the converter: edge detectors and wires of the graphical bodies
    _w1, _w2, _w3, _w4, _w5, _w6, _w7, _w8 : BOOL;
END_VAR

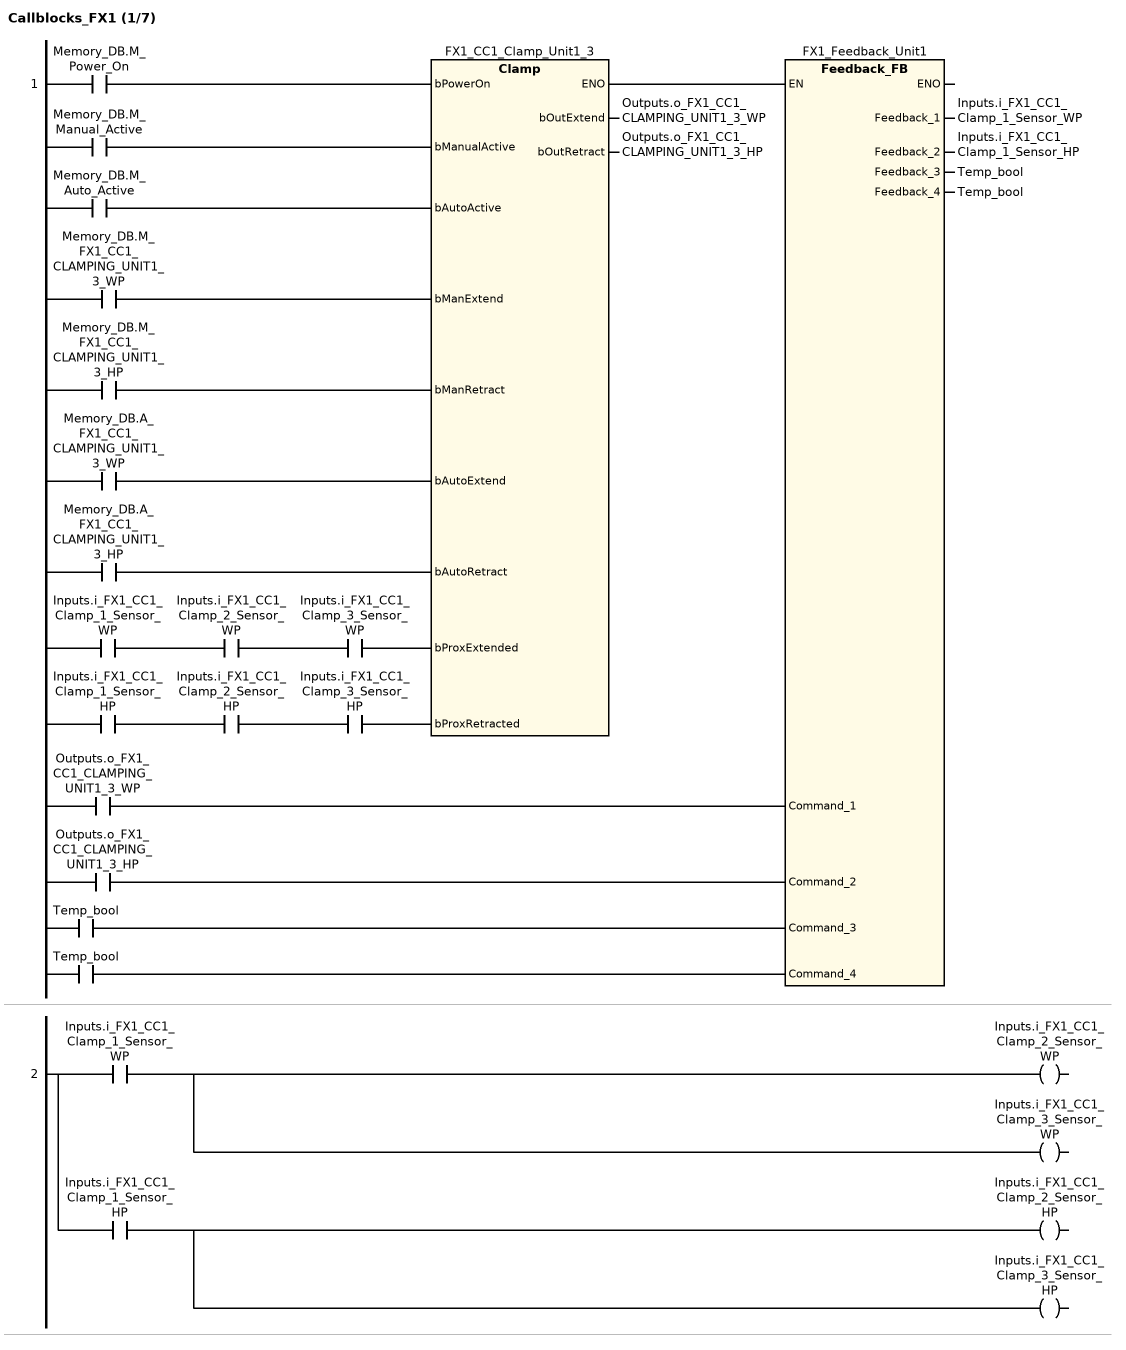
// NETWORK 1
FX1_CC1_Clamp_Unit1_3(
    bPowerOn := Memory_DB.M_Power_On,
    bManualActive := Memory_DB.M_Manual_Active,
    bAutoActive := Memory_DB.M_Auto_Active,
    bManExtend := Memory_DB.M_FX1_CC1_CLAMPING_UNIT1_3_WP,
    bManRetract := Memory_DB.M_FX1_CC1_CLAMPING_UNIT1_3_HP,
    bAutoExtend := Memory_DB.A_FX1_CC1_CLAMPING_UNIT1_3_WP,
    bAutoRetract := Memory_DB.A_FX1_CC1_CLAMPING_UNIT1_3_HP,
    bProxExtended := Inputs.i_FX1_CC1_Clamp_1_Sensor_WP AND Inputs.i_FX1_CC1_Clamp_2_Sensor_WP AND Inputs.i_FX1_CC1_Clamp_3_Sensor_WP,
    bProxRetracted := Inputs.i_FX1_CC1_Clamp_1_Sensor_HP AND Inputs.i_FX1_CC1_Clamp_2_Sensor_HP AND Inputs.i_FX1_CC1_Clamp_3_Sensor_HP,
    bOutExtend => Outputs.o_FX1_CC1_CLAMPING_UNIT1_3_WP,
    bOutRetract => Outputs.o_FX1_CC1_CLAMPING_UNIT1_3_HP); // Clamp
FX1_Feedback_Unit1(
    EN := TRUE,
    Command_1 := Outputs.o_FX1_CC1_CLAMPING_UNIT1_3_WP,
    Command_2 := Outputs.o_FX1_CC1_CLAMPING_UNIT1_3_HP,
    Command_3 := Temp_bool,
    Command_4 := Temp_bool,
    Feedback_1 => Inputs.i_FX1_CC1_Clamp_1_Sensor_WP,
    Feedback_2 => Inputs.i_FX1_CC1_Clamp_1_Sensor_HP,
    Feedback_3 => Temp_bool,
    Feedback_4 => Temp_bool); // Feedback_FB

// NETWORK 2
_w1 := Inputs.i_FX1_CC1_Clamp_1_Sensor_WP;
Inputs.i_FX1_CC1_Clamp_2_Sensor_WP := _w1;
Inputs.i_FX1_CC1_Clamp_3_Sensor_WP := _w1;
_w2 := Inputs.i_FX1_CC1_Clamp_1_Sensor_HP;
Inputs.i_FX1_CC1_Clamp_2_Sensor_HP := _w2;
Inputs.i_FX1_CC1_Clamp_3_Sensor_HP := _w2;

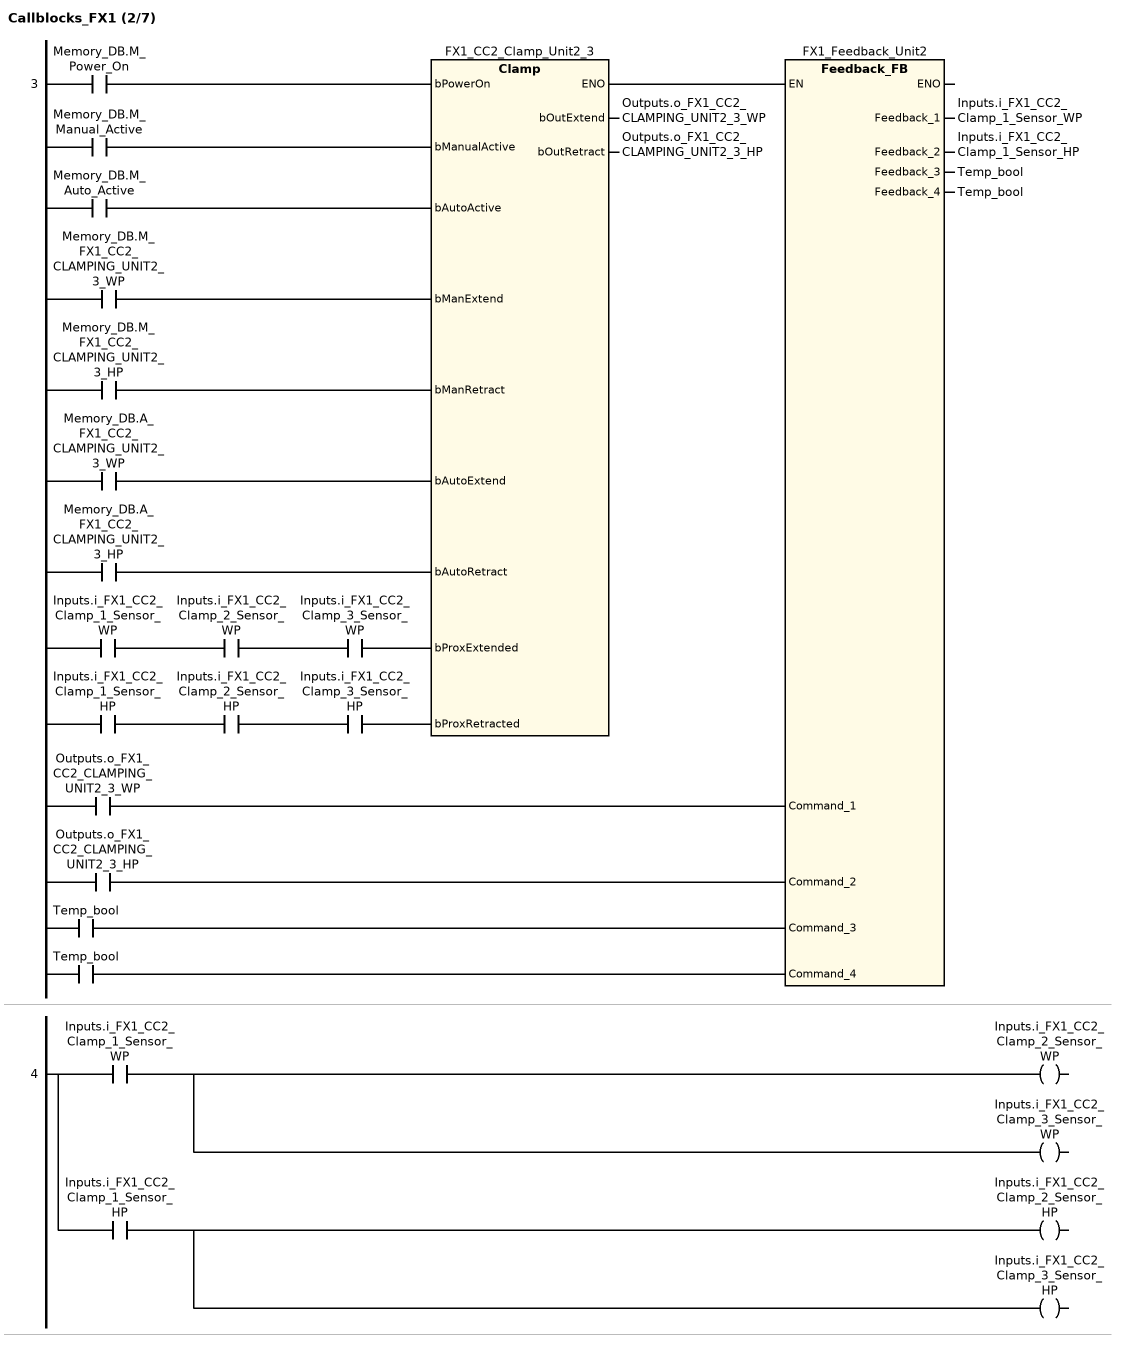
// NETWORK 3
FX1_CC2_Clamp_Unit2_3(
    bPowerOn := Memory_DB.M_Power_On,
    bManualActive := Memory_DB.M_Manual_Active,
    bAutoActive := Memory_DB.M_Auto_Active,
    bManExtend := Memory_DB.M_FX1_CC2_CLAMPING_UNIT2_3_WP,
    bManRetract := Memory_DB.M_FX1_CC2_CLAMPING_UNIT2_3_HP,
    bAutoExtend := Memory_DB.A_FX1_CC2_CLAMPING_UNIT2_3_WP,
    bAutoRetract := Memory_DB.A_FX1_CC2_CLAMPING_UNIT2_3_HP,
    bProxExtended := Inputs.i_FX1_CC2_Clamp_1_Sensor_WP AND Inputs.i_FX1_CC2_Clamp_2_Sensor_WP AND Inputs.i_FX1_CC2_Clamp_3_Sensor_WP,
    bProxRetracted := Inputs.i_FX1_CC2_Clamp_1_Sensor_HP AND Inputs.i_FX1_CC2_Clamp_2_Sensor_HP AND Inputs.i_FX1_CC2_Clamp_3_Sensor_HP,
    bOutExtend => Outputs.o_FX1_CC2_CLAMPING_UNIT2_3_WP,
    bOutRetract => Outputs.o_FX1_CC2_CLAMPING_UNIT2_3_HP); // Clamp
FX1_Feedback_Unit2(
    EN := TRUE,
    Command_1 := Outputs.o_FX1_CC2_CLAMPING_UNIT2_3_WP,
    Command_2 := Outputs.o_FX1_CC2_CLAMPING_UNIT2_3_HP,
    Command_3 := Temp_bool,
    Command_4 := Temp_bool,
    Feedback_1 => Inputs.i_FX1_CC2_Clamp_1_Sensor_WP,
    Feedback_2 => Inputs.i_FX1_CC2_Clamp_1_Sensor_HP,
    Feedback_3 => Temp_bool,
    Feedback_4 => Temp_bool); // Feedback_FB

// NETWORK 4
_w3 := Inputs.i_FX1_CC2_Clamp_1_Sensor_WP;
Inputs.i_FX1_CC2_Clamp_2_Sensor_WP := _w3;
Inputs.i_FX1_CC2_Clamp_3_Sensor_WP := _w3;
_w4 := Inputs.i_FX1_CC2_Clamp_1_Sensor_HP;
Inputs.i_FX1_CC2_Clamp_2_Sensor_HP := _w4;
Inputs.i_FX1_CC2_Clamp_3_Sensor_HP := _w4;

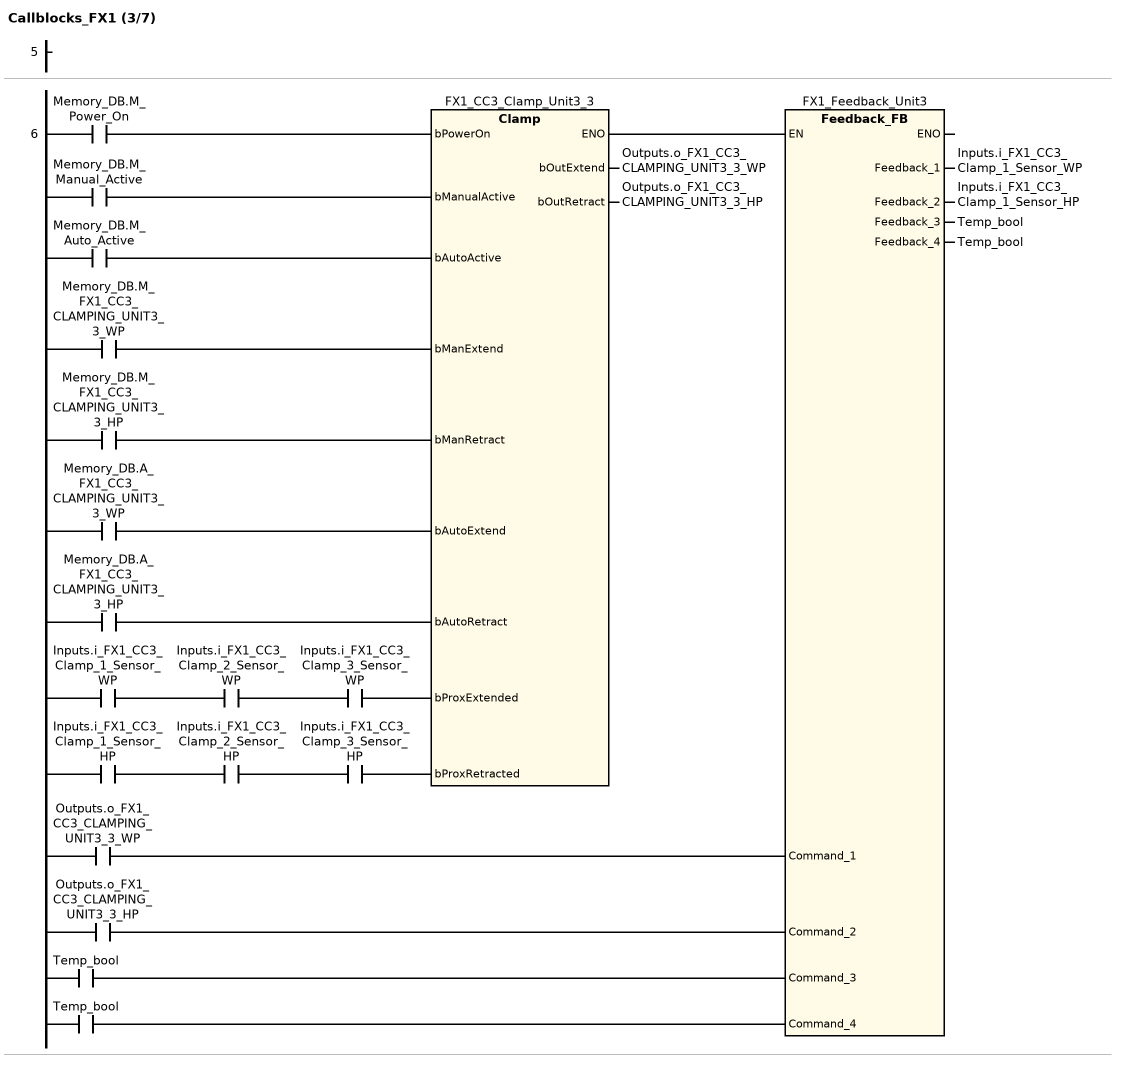
// NETWORK 5

// NETWORK 6
FX1_CC3_Clamp_Unit3_3(
    bPowerOn := Memory_DB.M_Power_On,
    bManualActive := Memory_DB.M_Manual_Active,
    bAutoActive := Memory_DB.M_Auto_Active,
    bManExtend := Memory_DB.M_FX1_CC3_CLAMPING_UNIT3_3_WP,
    bManRetract := Memory_DB.M_FX1_CC3_CLAMPING_UNIT3_3_HP,
    bAutoExtend := Memory_DB.A_FX1_CC3_CLAMPING_UNIT3_3_WP,
    bAutoRetract := Memory_DB.A_FX1_CC3_CLAMPING_UNIT3_3_HP,
    bProxExtended := Inputs.i_FX1_CC3_Clamp_1_Sensor_WP AND Inputs.i_FX1_CC3_Clamp_2_Sensor_WP AND Inputs.i_FX1_CC3_Clamp_3_Sensor_WP,
    bProxRetracted := Inputs.i_FX1_CC3_Clamp_1_Sensor_HP AND Inputs.i_FX1_CC3_Clamp_2_Sensor_HP AND Inputs.i_FX1_CC3_Clamp_3_Sensor_HP,
    bOutExtend => Outputs.o_FX1_CC3_CLAMPING_UNIT3_3_WP,
    bOutRetract => Outputs.o_FX1_CC3_CLAMPING_UNIT3_3_HP); // Clamp
FX1_Feedback_Unit3(
    EN := TRUE,
    Command_1 := Outputs.o_FX1_CC3_CLAMPING_UNIT3_3_WP,
    Command_2 := Outputs.o_FX1_CC3_CLAMPING_UNIT3_3_HP,
    Command_3 := Temp_bool,
    Command_4 := Temp_bool,
    Feedback_1 => Inputs.i_FX1_CC3_Clamp_1_Sensor_WP,
    Feedback_2 => Inputs.i_FX1_CC3_Clamp_1_Sensor_HP,
    Feedback_3 => Temp_bool,
    Feedback_4 => Temp_bool); // Feedback_FB

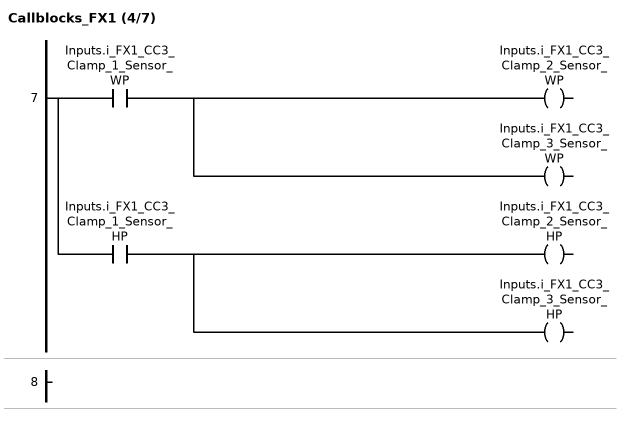
// NETWORK 7
_w5 := Inputs.i_FX1_CC3_Clamp_1_Sensor_WP;
Inputs.i_FX1_CC3_Clamp_2_Sensor_WP := _w5;
Inputs.i_FX1_CC3_Clamp_3_Sensor_WP := _w5;
_w6 := Inputs.i_FX1_CC3_Clamp_1_Sensor_HP;
Inputs.i_FX1_CC3_Clamp_2_Sensor_HP := _w6;
Inputs.i_FX1_CC3_Clamp_3_Sensor_HP := _w6;

// NETWORK 8

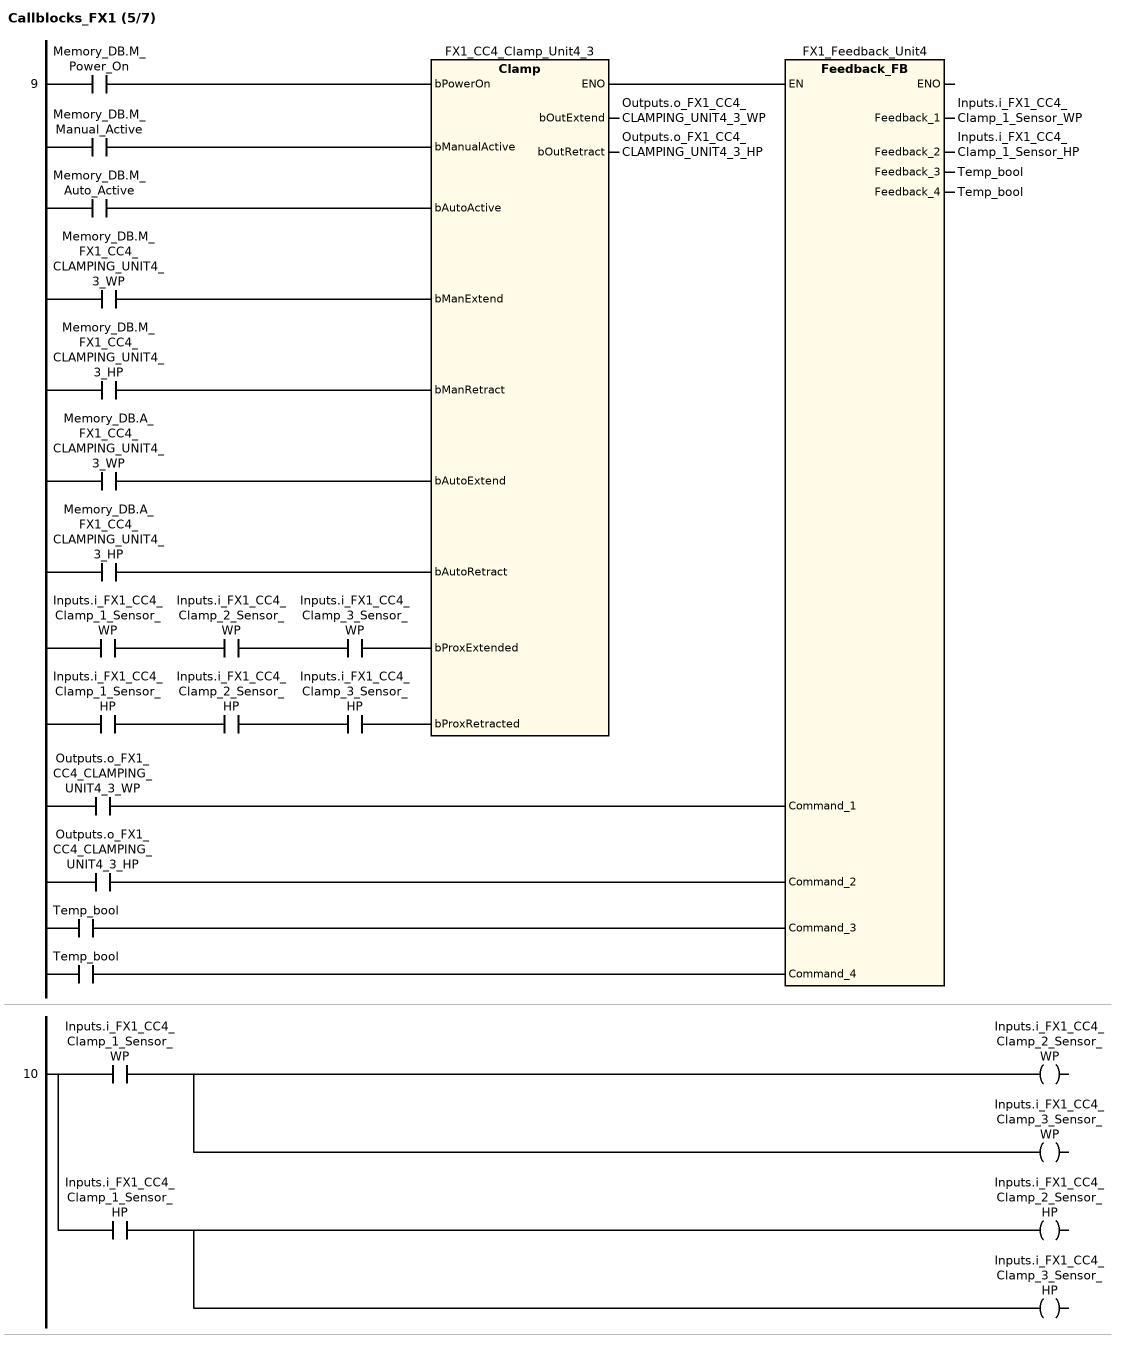
// NETWORK 9
FX1_CC4_Clamp_Unit4_3(
    bPowerOn := Memory_DB.M_Power_On,
    bManualActive := Memory_DB.M_Manual_Active,
    bAutoActive := Memory_DB.M_Auto_Active,
    bManExtend := Memory_DB.M_FX1_CC4_CLAMPING_UNIT4_3_WP,
    bManRetract := Memory_DB.M_FX1_CC4_CLAMPING_UNIT4_3_HP,
    bAutoExtend := Memory_DB.A_FX1_CC4_CLAMPING_UNIT4_3_WP,
    bAutoRetract := Memory_DB.A_FX1_CC4_CLAMPING_UNIT4_3_HP,
    bProxExtended := Inputs.i_FX1_CC4_Clamp_1_Sensor_WP AND Inputs.i_FX1_CC4_Clamp_2_Sensor_WP AND Inputs.i_FX1_CC4_Clamp_3_Sensor_WP,
    bProxRetracted := Inputs.i_FX1_CC4_Clamp_1_Sensor_HP AND Inputs.i_FX1_CC4_Clamp_2_Sensor_HP AND Inputs.i_FX1_CC4_Clamp_3_Sensor_HP,
    bOutExtend => Outputs.o_FX1_CC4_CLAMPING_UNIT4_3_WP,
    bOutRetract => Outputs.o_FX1_CC4_CLAMPING_UNIT4_3_HP); // Clamp
FX1_Feedback_Unit4(
    EN := TRUE,
    Command_1 := Outputs.o_FX1_CC4_CLAMPING_UNIT4_3_WP,
    Command_2 := Outputs.o_FX1_CC4_CLAMPING_UNIT4_3_HP,
    Command_3 := Temp_bool,
    Command_4 := Temp_bool,
    Feedback_1 => Inputs.i_FX1_CC4_Clamp_1_Sensor_WP,
    Feedback_2 => Inputs.i_FX1_CC4_Clamp_1_Sensor_HP,
    Feedback_3 => Temp_bool,
    Feedback_4 => Temp_bool); // Feedback_FB

// NETWORK 10
_w7 := Inputs.i_FX1_CC4_Clamp_1_Sensor_WP;
Inputs.i_FX1_CC4_Clamp_2_Sensor_WP := _w7;
Inputs.i_FX1_CC4_Clamp_3_Sensor_WP := _w7;
_w8 := Inputs.i_FX1_CC4_Clamp_1_Sensor_HP;
Inputs.i_FX1_CC4_Clamp_2_Sensor_HP := _w8;
Inputs.i_FX1_CC4_Clamp_3_Sensor_HP := _w8;

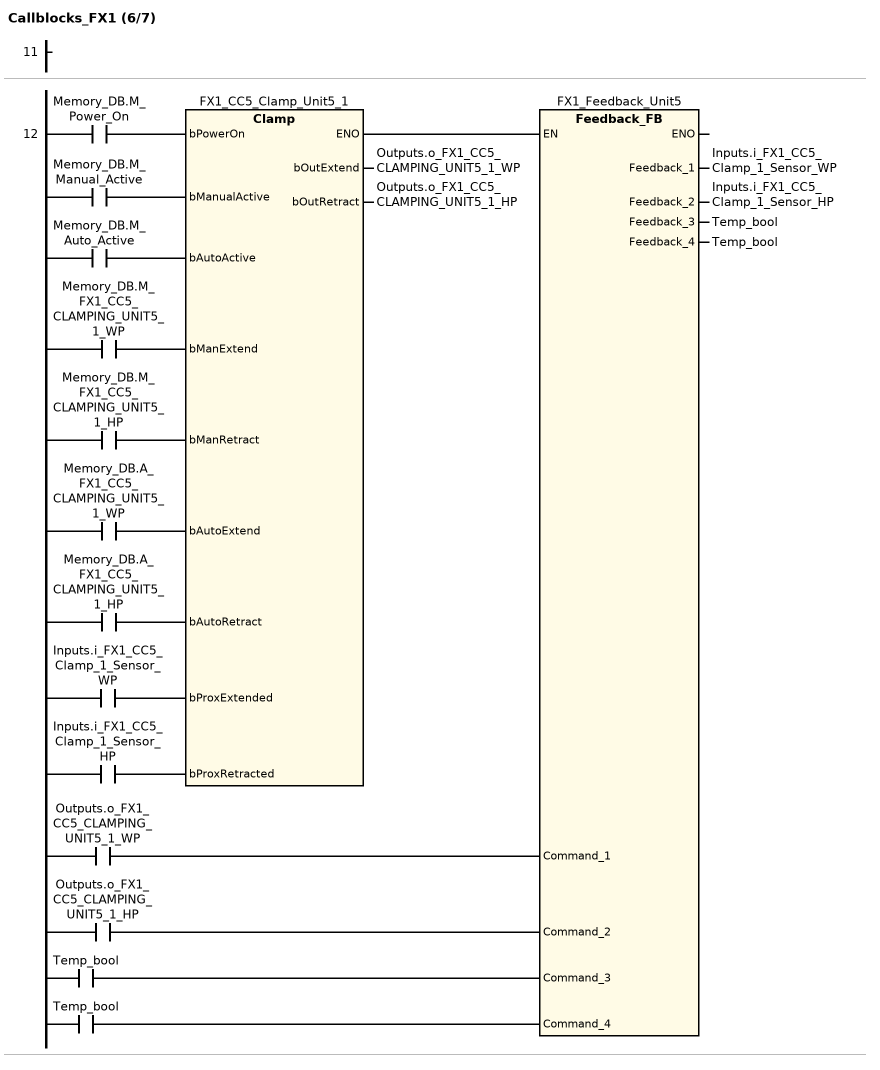
// NETWORK 11

// NETWORK 12
FX1_CC5_Clamp_Unit5_1(
    bPowerOn := Memory_DB.M_Power_On,
    bManualActive := Memory_DB.M_Manual_Active,
    bAutoActive := Memory_DB.M_Auto_Active,
    bManExtend := Memory_DB.M_FX1_CC5_CLAMPING_UNIT5_1_WP,
    bManRetract := Memory_DB.M_FX1_CC5_CLAMPING_UNIT5_1_HP,
    bAutoExtend := Memory_DB.A_FX1_CC5_CLAMPING_UNIT5_1_WP,
    bAutoRetract := Memory_DB.A_FX1_CC5_CLAMPING_UNIT5_1_HP,
    bProxExtended := Inputs.i_FX1_CC5_Clamp_1_Sensor_WP,
    bProxRetracted := Inputs.i_FX1_CC5_Clamp_1_Sensor_HP,
    bOutExtend => Outputs.o_FX1_CC5_CLAMPING_UNIT5_1_WP,
    bOutRetract => Outputs.o_FX1_CC5_CLAMPING_UNIT5_1_HP); // Clamp
FX1_Feedback_Unit5(
    EN := TRUE,
    Command_1 := Outputs.o_FX1_CC5_CLAMPING_UNIT5_1_WP,
    Command_2 := Outputs.o_FX1_CC5_CLAMPING_UNIT5_1_HP,
    Command_3 := Temp_bool,
    Command_4 := Temp_bool,
    Feedback_1 => Inputs.i_FX1_CC5_Clamp_1_Sensor_WP,
    Feedback_2 => Inputs.i_FX1_CC5_Clamp_1_Sensor_HP,
    Feedback_3 => Temp_bool,
    Feedback_4 => Temp_bool); // Feedback_FB

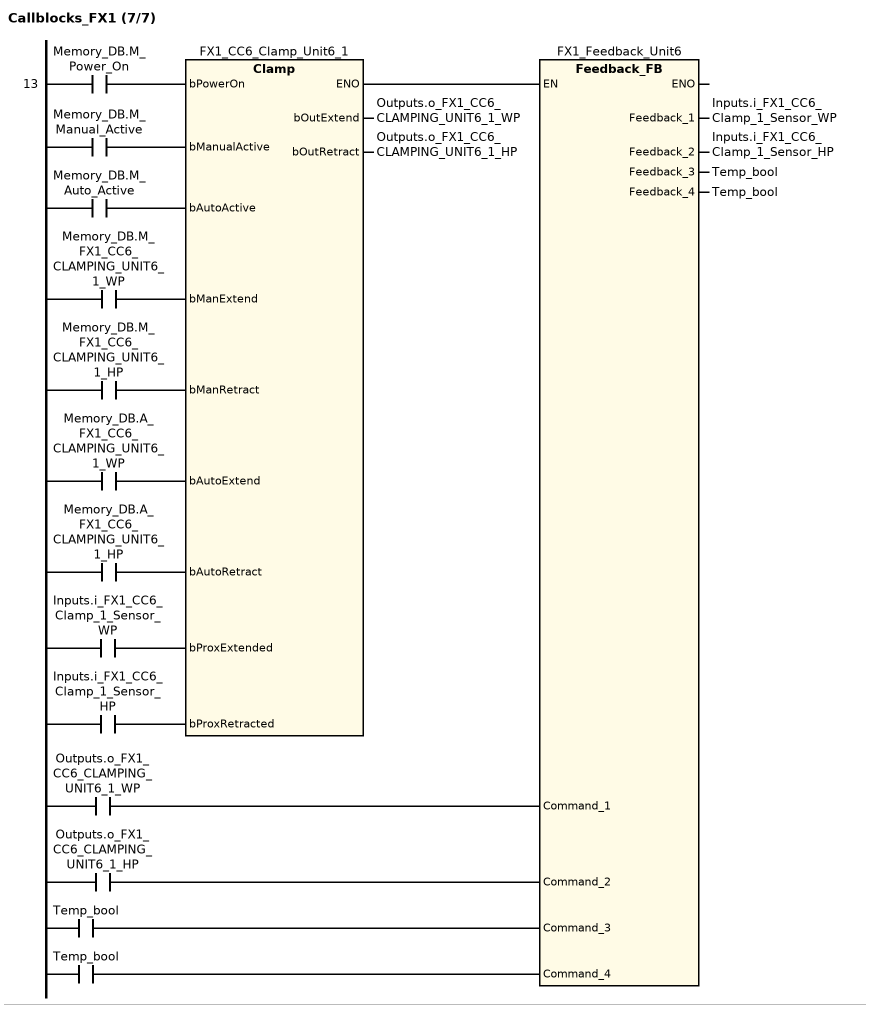
// NETWORK 13
FX1_CC6_Clamp_Unit6_1(
    bPowerOn := Memory_DB.M_Power_On,
    bManualActive := Memory_DB.M_Manual_Active,
    bAutoActive := Memory_DB.M_Auto_Active,
    bManExtend := Memory_DB.M_FX1_CC6_CLAMPING_UNIT6_1_WP,
    bManRetract := Memory_DB.M_FX1_CC6_CLAMPING_UNIT6_1_HP,
    bAutoExtend := Memory_DB.A_FX1_CC6_CLAMPING_UNIT6_1_WP,
    bAutoRetract := Memory_DB.A_FX1_CC6_CLAMPING_UNIT6_1_HP,
    bProxExtended := Inputs.i_FX1_CC6_Clamp_1_Sensor_WP,
    bProxRetracted := Inputs.i_FX1_CC6_Clamp_1_Sensor_HP,
    bOutExtend => Outputs.o_FX1_CC6_CLAMPING_UNIT6_1_WP,
    bOutRetract => Outputs.o_FX1_CC6_CLAMPING_UNIT6_1_HP); // Clamp
FX1_Feedback_Unit6(
    EN := TRUE,
    Command_1 := Outputs.o_FX1_CC6_CLAMPING_UNIT6_1_WP,
    Command_2 := Outputs.o_FX1_CC6_CLAMPING_UNIT6_1_HP,
    Command_3 := Temp_bool,
    Command_4 := Temp_bool,
    Feedback_1 => Inputs.i_FX1_CC6_Clamp_1_Sensor_WP,
    Feedback_2 => Inputs.i_FX1_CC6_Clamp_1_Sensor_HP,
    Feedback_3 => Temp_bool,
    Feedback_4 => Temp_bool); // Feedback_FB

END_PROGRAM

// ---- POUs/Callblocks_FX2.TcPOU
PROGRAM Callblocks_FX2
VAR

FX2_CC1_Clamp_Unit1_3 : clamp;
FX2_CC2_Clamp_Unit2_3 : clamp;
FX2_CC3_Clamp_Unit3_3 : clamp;
FX2_CC4_Clamp_Unit4_3 : clamp;
FX2_CC5_Clamp_Unit5_1 : clamp;
FX2_CC6_Clamp_Unit6_1 : clamp;

Temp_bool : BOOL;
FX2_Feedback_Unit1  : Feedback_FB;
FX2_Feedback_Unit2  : Feedback_FB;
FX2_Feedback_Unit3  : Feedback_FB;
FX2_Feedback_Unit4  : Feedback_FB;
FX2_Feedback_Unit5  : Feedback_FB;
FX2_Feedback_Unit6  : Feedback_FB;	

END_VAR
VAR // added by the converter: edge detectors and wires of the graphical bodies
    _w1, _w2, _w3, _w4, _w5, _w6, _w7, _w8 : BOOL;
END_VAR

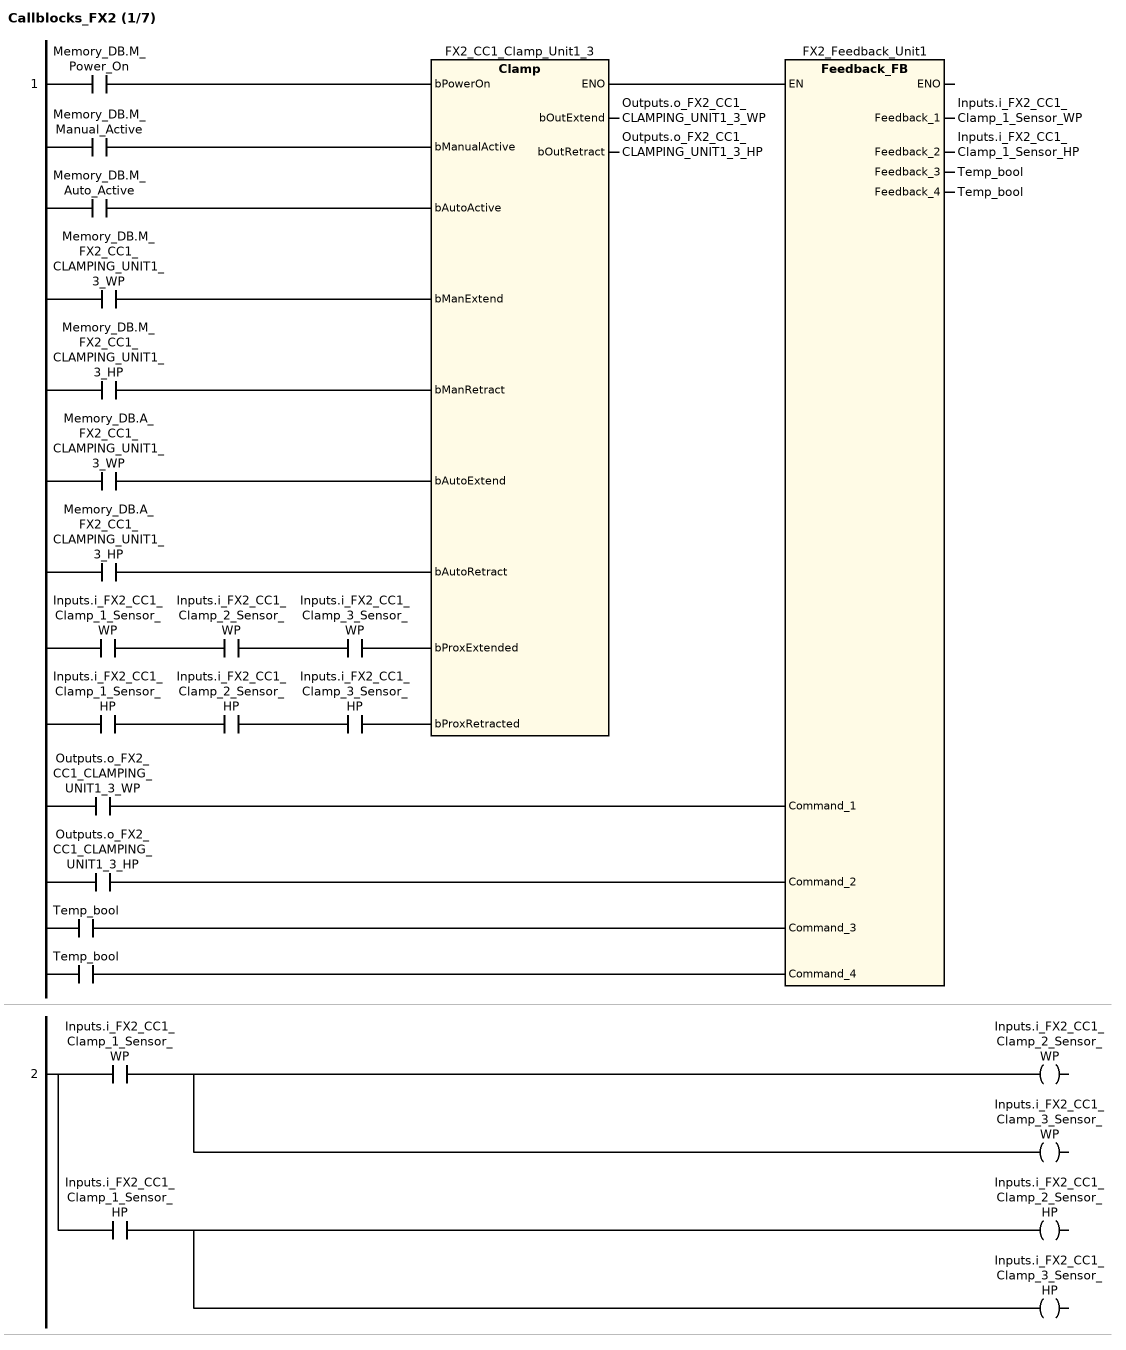
// NETWORK 1
FX2_CC1_Clamp_Unit1_3(
    bPowerOn := Memory_DB.M_Power_On,
    bManualActive := Memory_DB.M_Manual_Active,
    bAutoActive := Memory_DB.M_Auto_Active,
    bManExtend := Memory_DB.M_FX2_CC1_CLAMPING_UNIT1_3_WP,
    bManRetract := Memory_DB.M_FX2_CC1_CLAMPING_UNIT1_3_HP,
    bAutoExtend := Memory_DB.A_FX2_CC1_CLAMPING_UNIT1_3_WP,
    bAutoRetract := Memory_DB.A_FX2_CC1_CLAMPING_UNIT1_3_HP,
    bProxExtended := Inputs.i_FX2_CC1_Clamp_1_Sensor_WP AND Inputs.i_FX2_CC1_Clamp_2_Sensor_WP AND Inputs.i_FX2_CC1_Clamp_3_Sensor_WP,
    bProxRetracted := Inputs.i_FX2_CC1_Clamp_1_Sensor_HP AND Inputs.i_FX2_CC1_Clamp_2_Sensor_HP AND Inputs.i_FX2_CC1_Clamp_3_Sensor_HP,
    bOutExtend => Outputs.o_FX2_CC1_CLAMPING_UNIT1_3_WP,
    bOutRetract => Outputs.o_FX2_CC1_CLAMPING_UNIT1_3_HP); // Clamp
FX2_Feedback_Unit1(
    EN := TRUE,
    Command_1 := Outputs.o_FX2_CC1_CLAMPING_UNIT1_3_WP,
    Command_2 := Outputs.o_FX2_CC1_CLAMPING_UNIT1_3_HP,
    Command_3 := Temp_bool,
    Command_4 := Temp_bool,
    Feedback_1 => Inputs.i_FX2_CC1_Clamp_1_Sensor_WP,
    Feedback_2 => Inputs.i_FX2_CC1_Clamp_1_Sensor_HP,
    Feedback_3 => Temp_bool,
    Feedback_4 => Temp_bool); // Feedback_FB

// NETWORK 2
_w1 := Inputs.i_FX2_CC1_Clamp_1_Sensor_WP;
Inputs.i_FX2_CC1_Clamp_2_Sensor_WP := _w1;
Inputs.i_FX2_CC1_Clamp_3_Sensor_WP := _w1;
_w2 := Inputs.i_FX2_CC1_Clamp_1_Sensor_HP;
Inputs.i_FX2_CC1_Clamp_2_Sensor_HP := _w2;
Inputs.i_FX2_CC1_Clamp_3_Sensor_HP := _w2;

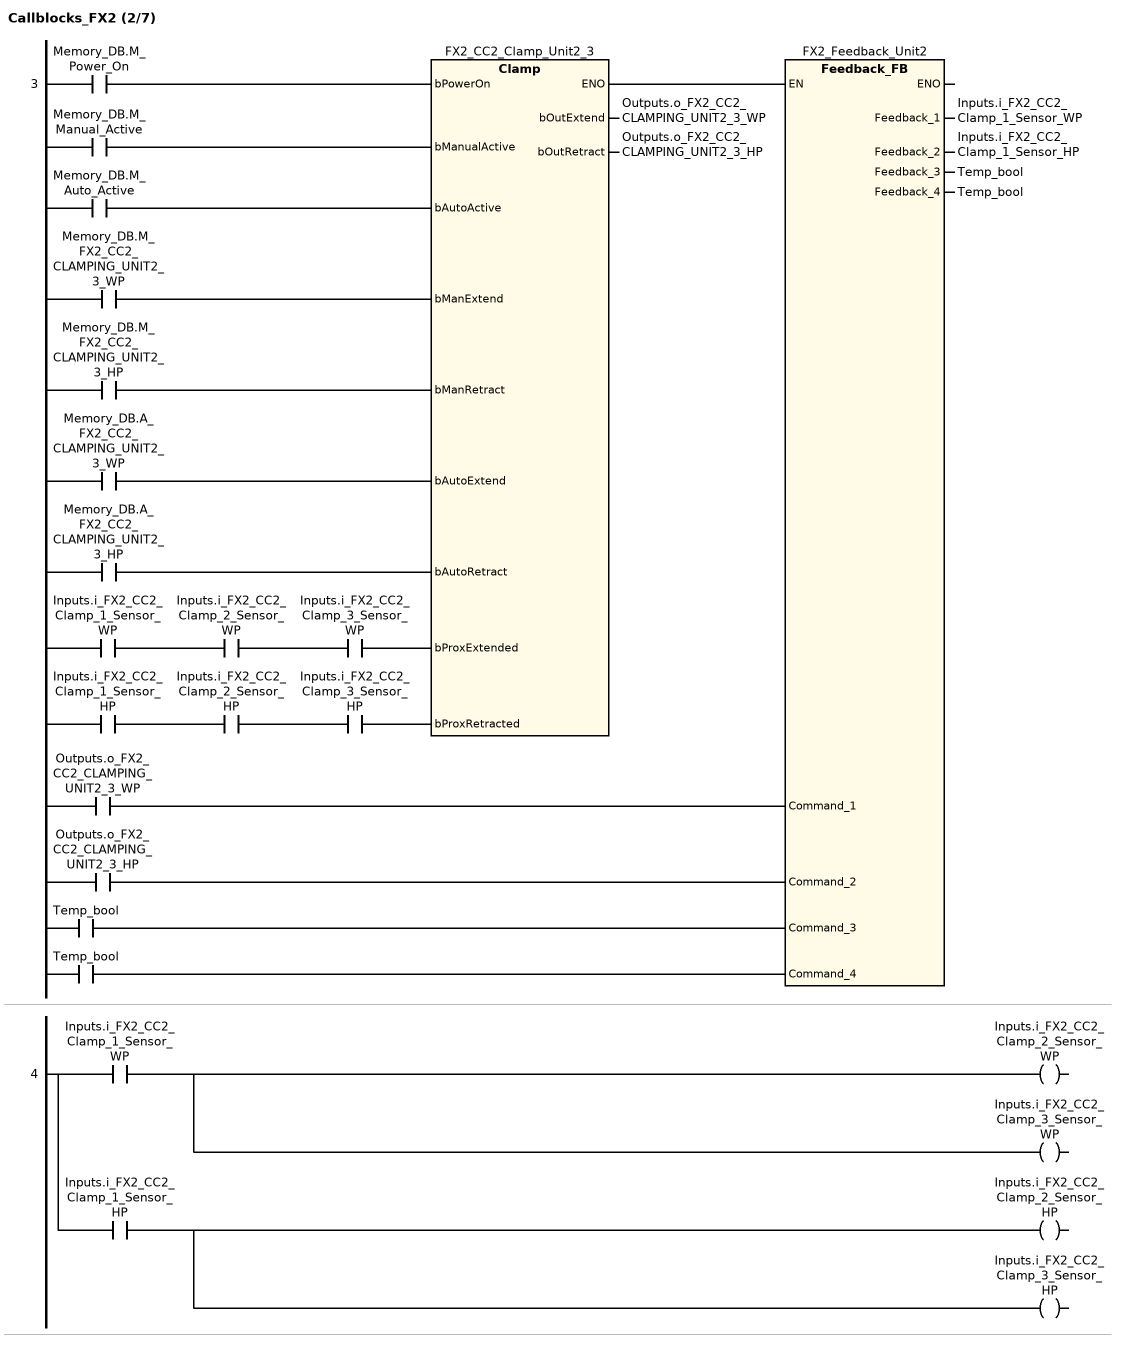
// NETWORK 3
FX2_CC2_Clamp_Unit2_3(
    bPowerOn := Memory_DB.M_Power_On,
    bManualActive := Memory_DB.M_Manual_Active,
    bAutoActive := Memory_DB.M_Auto_Active,
    bManExtend := Memory_DB.M_FX2_CC2_CLAMPING_UNIT2_3_WP,
    bManRetract := Memory_DB.M_FX2_CC2_CLAMPING_UNIT2_3_HP,
    bAutoExtend := Memory_DB.A_FX2_CC2_CLAMPING_UNIT2_3_WP,
    bAutoRetract := Memory_DB.A_FX2_CC2_CLAMPING_UNIT2_3_HP,
    bProxExtended := Inputs.i_FX2_CC2_Clamp_1_Sensor_WP AND Inputs.i_FX2_CC2_Clamp_2_Sensor_WP AND Inputs.i_FX2_CC2_Clamp_3_Sensor_WP,
    bProxRetracted := Inputs.i_FX2_CC2_Clamp_1_Sensor_HP AND Inputs.i_FX2_CC2_Clamp_2_Sensor_HP AND Inputs.i_FX2_CC2_Clamp_3_Sensor_HP,
    bOutExtend => Outputs.o_FX2_CC2_CLAMPING_UNIT2_3_WP,
    bOutRetract => Outputs.o_FX2_CC2_CLAMPING_UNIT2_3_HP); // Clamp
FX2_Feedback_Unit2(
    EN := TRUE,
    Command_1 := Outputs.o_FX2_CC2_CLAMPING_UNIT2_3_WP,
    Command_2 := Outputs.o_FX2_CC2_CLAMPING_UNIT2_3_HP,
    Command_3 := Temp_bool,
    Command_4 := Temp_bool,
    Feedback_1 => Inputs.i_FX2_CC2_Clamp_1_Sensor_WP,
    Feedback_2 => Inputs.i_FX2_CC2_Clamp_1_Sensor_HP,
    Feedback_3 => Temp_bool,
    Feedback_4 => Temp_bool); // Feedback_FB

// NETWORK 4
_w3 := Inputs.i_FX2_CC2_Clamp_1_Sensor_WP;
Inputs.i_FX2_CC2_Clamp_2_Sensor_WP := _w3;
Inputs.i_FX2_CC2_Clamp_3_Sensor_WP := _w3;
_w4 := Inputs.i_FX2_CC2_Clamp_1_Sensor_HP;
Inputs.i_FX2_CC2_Clamp_2_Sensor_HP := _w4;
Inputs.i_FX2_CC2_Clamp_3_Sensor_HP := _w4;

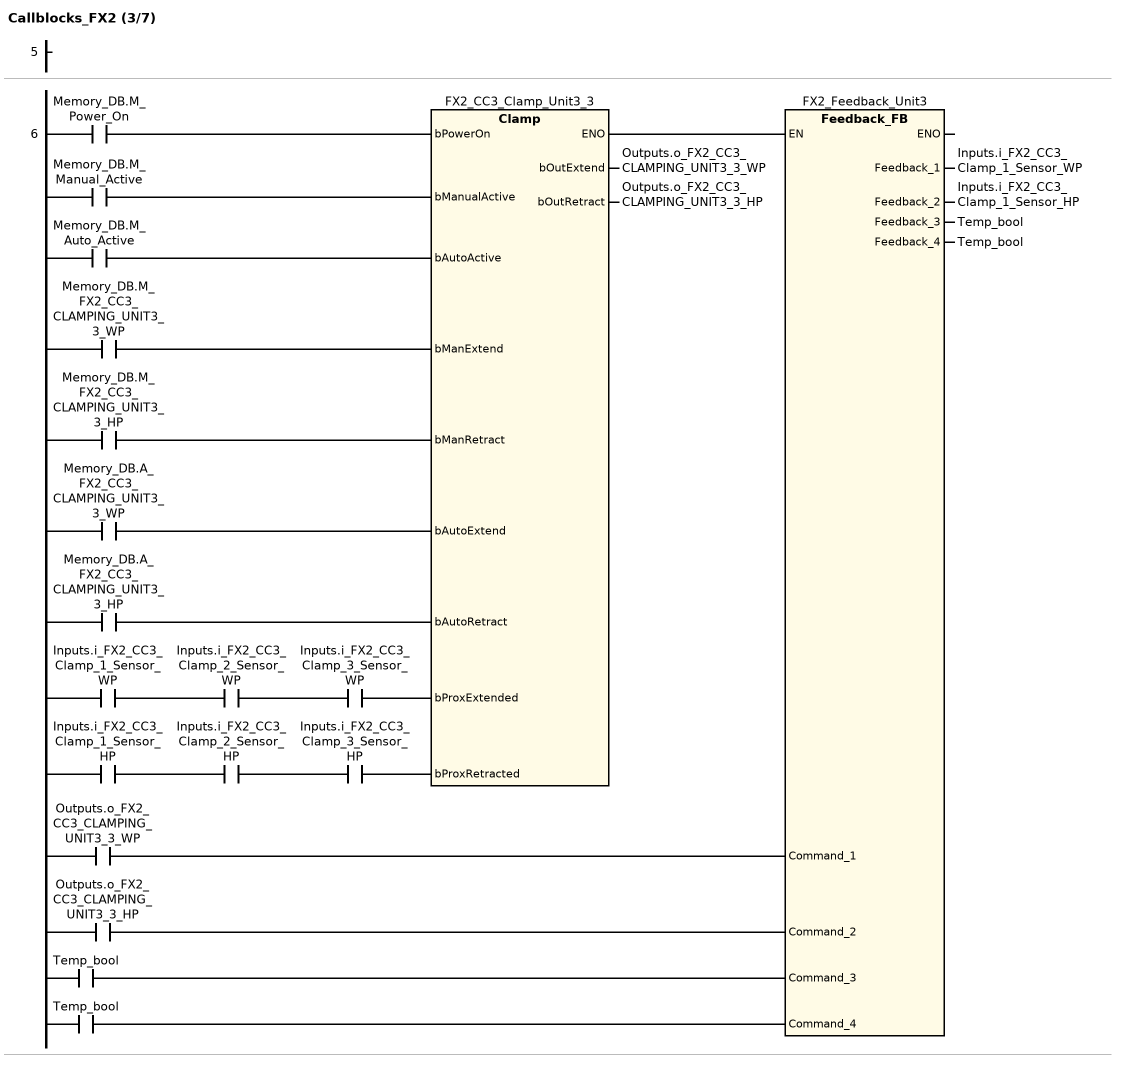
// NETWORK 5

// NETWORK 6
FX2_CC3_Clamp_Unit3_3(
    bPowerOn := Memory_DB.M_Power_On,
    bManualActive := Memory_DB.M_Manual_Active,
    bAutoActive := Memory_DB.M_Auto_Active,
    bManExtend := Memory_DB.M_FX2_CC3_CLAMPING_UNIT3_3_WP,
    bManRetract := Memory_DB.M_FX2_CC3_CLAMPING_UNIT3_3_HP,
    bAutoExtend := Memory_DB.A_FX2_CC3_CLAMPING_UNIT3_3_WP,
    bAutoRetract := Memory_DB.A_FX2_CC3_CLAMPING_UNIT3_3_HP,
    bProxExtended := Inputs.i_FX2_CC3_Clamp_1_Sensor_WP AND Inputs.i_FX2_CC3_Clamp_2_Sensor_WP AND Inputs.i_FX2_CC3_Clamp_3_Sensor_WP,
    bProxRetracted := Inputs.i_FX2_CC3_Clamp_1_Sensor_HP AND Inputs.i_FX2_CC3_Clamp_2_Sensor_HP AND Inputs.i_FX2_CC3_Clamp_3_Sensor_HP,
    bOutExtend => Outputs.o_FX2_CC3_CLAMPING_UNIT3_3_WP,
    bOutRetract => Outputs.o_FX2_CC3_CLAMPING_UNIT3_3_HP); // Clamp
FX2_Feedback_Unit3(
    EN := TRUE,
    Command_1 := Outputs.o_FX2_CC3_CLAMPING_UNIT3_3_WP,
    Command_2 := Outputs.o_FX2_CC3_CLAMPING_UNIT3_3_HP,
    Command_3 := Temp_bool,
    Command_4 := Temp_bool,
    Feedback_1 => Inputs.i_FX2_CC3_Clamp_1_Sensor_WP,
    Feedback_2 => Inputs.i_FX2_CC3_Clamp_1_Sensor_HP,
    Feedback_3 => Temp_bool,
    Feedback_4 => Temp_bool); // Feedback_FB

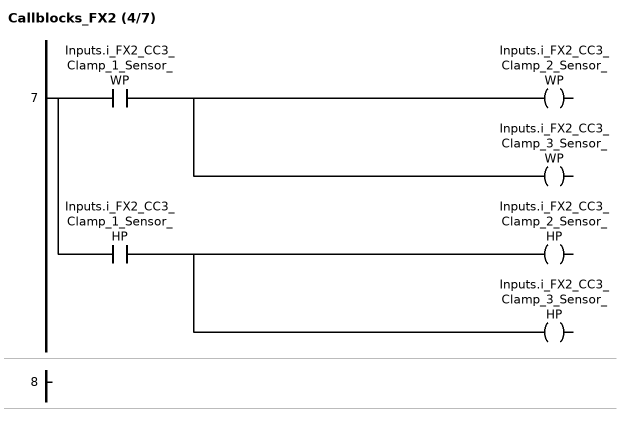
// NETWORK 7
_w5 := Inputs.i_FX2_CC3_Clamp_1_Sensor_WP;
Inputs.i_FX2_CC3_Clamp_2_Sensor_WP := _w5;
Inputs.i_FX2_CC3_Clamp_3_Sensor_WP := _w5;
_w6 := Inputs.i_FX2_CC3_Clamp_1_Sensor_HP;
Inputs.i_FX2_CC3_Clamp_2_Sensor_HP := _w6;
Inputs.i_FX2_CC3_Clamp_3_Sensor_HP := _w6;

// NETWORK 8

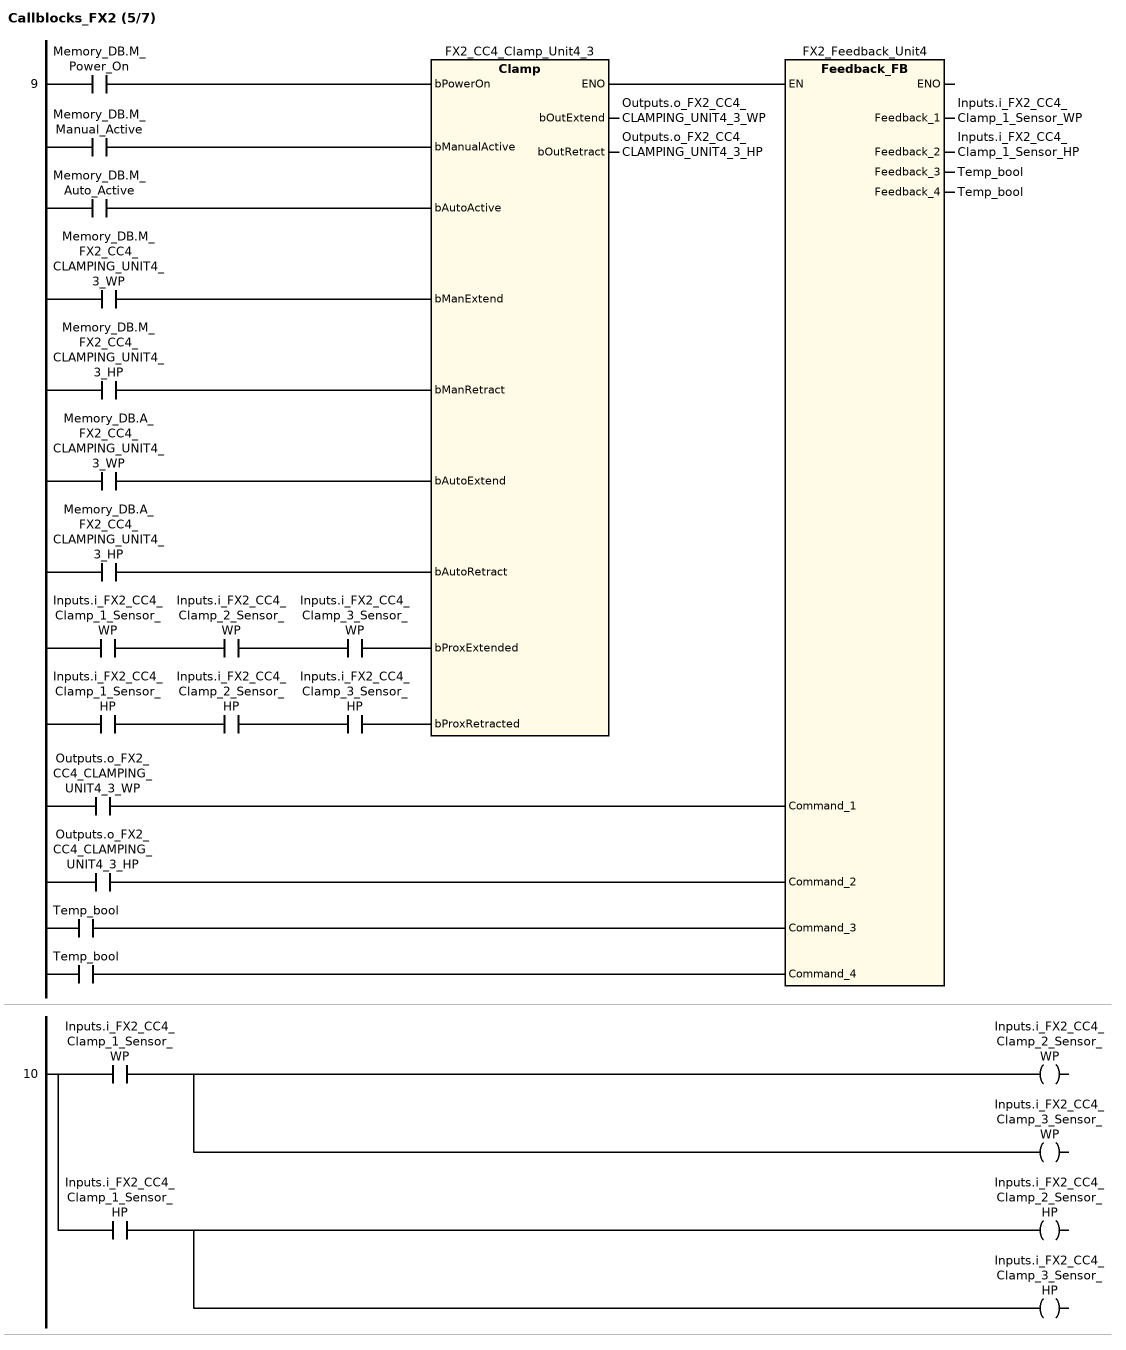
// NETWORK 9
FX2_CC4_Clamp_Unit4_3(
    bPowerOn := Memory_DB.M_Power_On,
    bManualActive := Memory_DB.M_Manual_Active,
    bAutoActive := Memory_DB.M_Auto_Active,
    bManExtend := Memory_DB.M_FX2_CC4_CLAMPING_UNIT4_3_WP,
    bManRetract := Memory_DB.M_FX2_CC4_CLAMPING_UNIT4_3_HP,
    bAutoExtend := Memory_DB.A_FX2_CC4_CLAMPING_UNIT4_3_WP,
    bAutoRetract := Memory_DB.A_FX2_CC4_CLAMPING_UNIT4_3_HP,
    bProxExtended := Inputs.i_FX2_CC4_Clamp_1_Sensor_WP AND Inputs.i_FX2_CC4_Clamp_2_Sensor_WP AND Inputs.i_FX2_CC4_Clamp_3_Sensor_WP,
    bProxRetracted := Inputs.i_FX2_CC4_Clamp_1_Sensor_HP AND Inputs.i_FX2_CC4_Clamp_2_Sensor_HP AND Inputs.i_FX2_CC4_Clamp_3_Sensor_HP,
    bOutExtend => Outputs.o_FX2_CC4_CLAMPING_UNIT4_3_WP,
    bOutRetract => Outputs.o_FX2_CC4_CLAMPING_UNIT4_3_HP); // Clamp
FX2_Feedback_Unit4(
    EN := TRUE,
    Command_1 := Outputs.o_FX2_CC4_CLAMPING_UNIT4_3_WP,
    Command_2 := Outputs.o_FX2_CC4_CLAMPING_UNIT4_3_HP,
    Command_3 := Temp_bool,
    Command_4 := Temp_bool,
    Feedback_1 => Inputs.i_FX2_CC4_Clamp_1_Sensor_WP,
    Feedback_2 => Inputs.i_FX2_CC4_Clamp_1_Sensor_HP,
    Feedback_3 => Temp_bool,
    Feedback_4 => Temp_bool); // Feedback_FB

// NETWORK 10
_w7 := Inputs.i_FX2_CC4_Clamp_1_Sensor_WP;
Inputs.i_FX2_CC4_Clamp_2_Sensor_WP := _w7;
Inputs.i_FX2_CC4_Clamp_3_Sensor_WP := _w7;
_w8 := Inputs.i_FX2_CC4_Clamp_1_Sensor_HP;
Inputs.i_FX2_CC4_Clamp_2_Sensor_HP := _w8;
Inputs.i_FX2_CC4_Clamp_3_Sensor_HP := _w8;

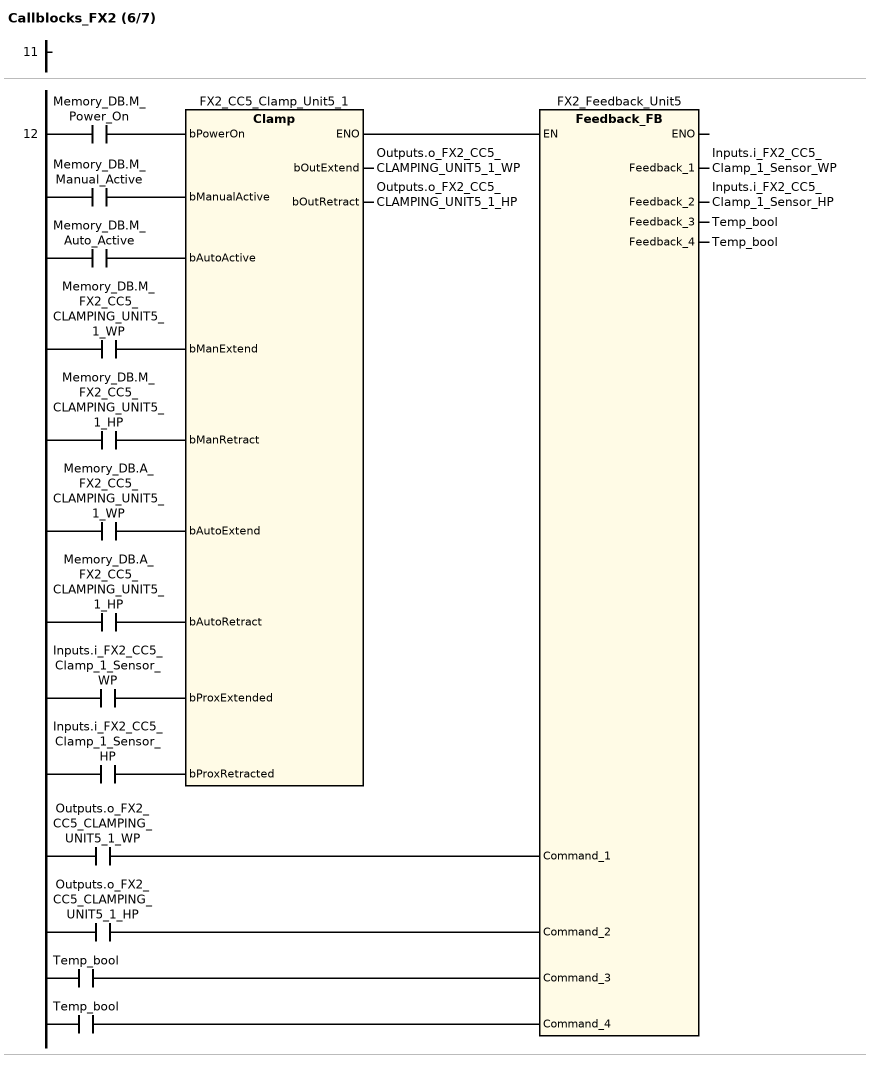
// NETWORK 11

// NETWORK 12
FX2_CC5_Clamp_Unit5_1(
    bPowerOn := Memory_DB.M_Power_On,
    bManualActive := Memory_DB.M_Manual_Active,
    bAutoActive := Memory_DB.M_Auto_Active,
    bManExtend := Memory_DB.M_FX2_CC5_CLAMPING_UNIT5_1_WP,
    bManRetract := Memory_DB.M_FX2_CC5_CLAMPING_UNIT5_1_HP,
    bAutoExtend := Memory_DB.A_FX2_CC5_CLAMPING_UNIT5_1_WP,
    bAutoRetract := Memory_DB.A_FX2_CC5_CLAMPING_UNIT5_1_HP,
    bProxExtended := Inputs.i_FX2_CC5_Clamp_1_Sensor_WP,
    bProxRetracted := Inputs.i_FX2_CC5_Clamp_1_Sensor_HP,
    bOutExtend => Outputs.o_FX2_CC5_CLAMPING_UNIT5_1_WP,
    bOutRetract => Outputs.o_FX2_CC5_CLAMPING_UNIT5_1_HP); // Clamp
FX2_Feedback_Unit5(
    EN := TRUE,
    Command_1 := Outputs.o_FX2_CC5_CLAMPING_UNIT5_1_WP,
    Command_2 := Outputs.o_FX2_CC5_CLAMPING_UNIT5_1_HP,
    Command_3 := Temp_bool,
    Command_4 := Temp_bool,
    Feedback_1 => Inputs.i_FX2_CC5_Clamp_1_Sensor_WP,
    Feedback_2 => Inputs.i_FX2_CC5_Clamp_1_Sensor_HP,
    Feedback_3 => Temp_bool,
    Feedback_4 => Temp_bool); // Feedback_FB

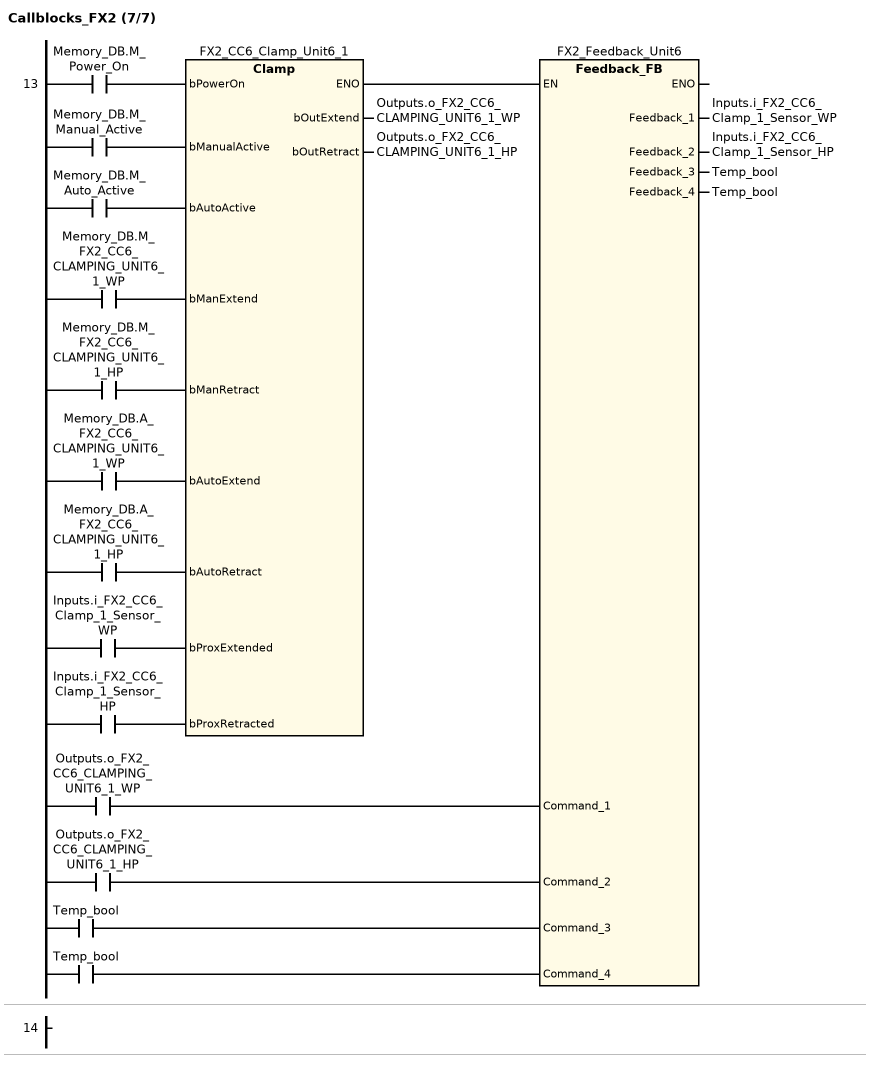
// NETWORK 13
FX2_CC6_Clamp_Unit6_1(
    bPowerOn := Memory_DB.M_Power_On,
    bManualActive := Memory_DB.M_Manual_Active,
    bAutoActive := Memory_DB.M_Auto_Active,
    bManExtend := Memory_DB.M_FX2_CC6_CLAMPING_UNIT6_1_WP,
    bManRetract := Memory_DB.M_FX2_CC6_CLAMPING_UNIT6_1_HP,
    bAutoExtend := Memory_DB.A_FX2_CC6_CLAMPING_UNIT6_1_WP,
    bAutoRetract := Memory_DB.A_FX2_CC6_CLAMPING_UNIT6_1_HP,
    bProxExtended := Inputs.i_FX2_CC6_Clamp_1_Sensor_WP,
    bProxRetracted := Inputs.i_FX2_CC6_Clamp_1_Sensor_HP,
    bOutExtend => Outputs.o_FX2_CC6_CLAMPING_UNIT6_1_WP,
    bOutRetract => Outputs.o_FX2_CC6_CLAMPING_UNIT6_1_HP); // Clamp
FX2_Feedback_Unit6(
    EN := TRUE,
    Command_1 := Outputs.o_FX2_CC6_CLAMPING_UNIT6_1_WP,
    Command_2 := Outputs.o_FX2_CC6_CLAMPING_UNIT6_1_HP,
    Command_3 := Temp_bool,
    Command_4 := Temp_bool,
    Feedback_1 => Inputs.i_FX2_CC6_Clamp_1_Sensor_WP,
    Feedback_2 => Inputs.i_FX2_CC6_Clamp_1_Sensor_HP,
    Feedback_3 => Temp_bool,
    Feedback_4 => Temp_bool); // Feedback_FB

// NETWORK 14

END_PROGRAM

// ---- GlobalTextList.TcGTLO
TEXTLIST GlobalTextList
  608 = ' Busy '
  896 = ' Job2 Done '
  971 = ' Pounce'
  134 = ' R01 Job Done '
  118 = ' R01 Job Done1 '
  143 = ' R01 Job Done2 '
  889 = ' R01 Job1 Done '
  932 = ' R01 Job2 Done '
  423 = ' R02 Busy '
  751 = ' R02 Home '
  374 = ' R02 Job Done '
  961 = ' R02 Job Done1 '
  517 = ' R02 Job Done2 '
  954 = ' R02 Job1 Done '
  725 = ' R02 Job2 Done '
  974 = ' R03 At Pounse'
  12 = ' R03 Drop Done '
  87 = ' R03 Drop1 Done '
  227 = ' R03 Drop2 Done '
  639 = ' R03 Pick1 Done '
  43 = ' R03 Pick2 Done '
  715 = '180 Deg'
  77 = '80 Deg'
  297 = 'Add'
  829 = 'All Safety Ok'
  834 = 'Auto'
  105 = 'Busy '
  368 = 'CC1 CLAMP'
  948 = 'CC1 CLAMP1'
  922 = 'CC1 CLAMP1-3'
  642 = 'CC2 CLAMP'
  179 = 'CC3 CLAMP'
  711 = 'CC4 CLAMP'
  151 = 'CC5 CLAMP'
  303 = 'CC6 CLAMP'
  910 = 'Cycle Start'
  207 = 'Cycle Start PB'
  388 = 'DOWN'
  146 = 'Down'
  152 = 'FD Down'
  566 = 'FD Up'
  527 = 'FIXTURE 1 MANUAL ACTION'
  946 = 'FIXTURE 2 MANUAL ACTION'
  451 = 'Fixture1 Load1'
  773 = 'Fixture1 Load1 Part Present'
  49 = 'Fixture1 Load2'
  590 = 'Fixture1 Load2 Part Present'
  835 = 'Fixture2 Load1'
  876 = 'Fixture2 Load1 Part Present'
  223 = 'Fixture2 Load2'
  236 = 'Fixture2 Load2 Part Present'
  275 = 'FR1 Load1 Part Present'
  246 = 'FRONT DOOR'
  551 = 'Front DR Closed'
  728 = 'Front DR Down'
  805 = 'Front DR Open'
  224 = 'Front DR Up'
  322 = 'FX1 Load1'
  414 = 'FX1 Load2'
  568 = 'FX1 TR -20 Deg'
  560 = 'FX1 TRUNION'
  492 = 'FX1TR-20 Deg'
  195 = 'FX2 Load1'
  125 = 'FX2 Load2'
  927 = 'FX2 TR -20 Deg'
  817 = 'FX2 TRUNION'
  1024 = 'FX2TR-20 Deg'
  645 = 'Home'
  824 = 'Initialise'
  641 = 'Initialised'
  858 = 'Job1 Done '
  166 = 'Job2 Done '
  504 = 'Manual'
  901 = 'MH R03 '
  897 = 'MH R03 Home '
  567 = 'Mode Selection'
  371 = 'Pick1 Done '
  632 = 'Pick2 Done '
  333 = 'Pos1'
  580 = 'Pos2'
  569 = 'Power ON PB'
  3 = 'Power On PB'
  748 = 'R01 Busy '
  940 = 'R01 Home '
  926 = 'R03 At Pounce'
  185 = 'R03 At Pounse'
  292 = 'R03 Home '
  193 = 'Rare DR Down'
  849 = 'Rare DR Up'
  37 = 'RD Down'
  422 = 'RD Up'
  602 = 'REAR DOOR'
  918 = 'Rear DR Down'
  404 = 'Rear DR Up'
  263 = 'Safety Ok'
  192 = 'Seq Init'
  505 = 'Seq Initialise'
  956 = 'Seq Int'
  23 = 'Start PB'
  426 = 'Stop PB'
  438 = 'TR At -20 Deg'
  141 = 'TR At 20 Deg'
  913 = 'TR At 80 Deg'
  730 = 'TT 0 Deg'
  555 = 'TT AT 0 Deg'
  589 = 'TT At 0 Deg'
  111 = 'TT AT 180 Deg'
  949 = 'TT At 180 Deg'
  369 = 'TURNTABLE'
  707 = 'UP'
  955 = 'Up'
  304 = 'Weld R01 Home '
  44 = 'Weld R01 Job Done '
  498 = 'Weld R02 Home '
  935 = 'Work'
END_TEXTLIST

// ---- POUs/FX2TextList.TcTLO
TEXTLIST FX2TextList
  0 = 'Wait For Fixture Home Pos &  Front Door Open'
  10 = 'Wait For Load1 complete & Door Closed'
  20 = 'Wait For Fixture Clamps Closed '
  30 = 'Wait for Trunion move to Pos2'
  40 = 'Wait for Front Door Open for Second load'
  50 = 'Wait for Load2 Complete & Door Closed'
  60 = 'Wait For Fixture Clamps Closed '
  70 = 'Wait For Trunion move to Pos1 '
  80 = 'Wait for Turntable to move Work Pos'
  90 = 'Wait for Weld Start Cmd to R1 & R2 Robot for First Weld'
  100 = 'Wait for Trunion move to Pos2'
  110 = 'Wait for Weld Start Cmd to R1 & R2 Robot for Second Weld'
  120 = 'Wait For Trunion move to Pos1 For Unload '
  130 = 'Wait For Rear Door Open'
  140 = 'Wait for Unload Start Cmd for R3 Robot'
  150 = 'Wait For Fixture Clamps Opened '
  160 = 'Wait for R3 Robot Pick 1 Complete'
  170 = 'Wait for R3 Robot Move to Pounce'
  180 = 'Wait for Trunion move to Pos2'
  190 = 'Wait For Fixture Clamps Opened '
  200 = 'Wait for R3 Robot Pick 2 Complete'
  210 = 'Wait for Trunion move to Pos1'
  220 = 'Wait For Rear Door Closed'
  230 = 'Wait for R3 Robot Drop 1 Complete'
  240 = 'Wait for R3 Robot Drop 2 Complete'
  250 = 'Wait for Tuntable Rotate to Load Position'
   = ''
END_TEXTLIST

// ---- POUs/FX1TextList.TcTLO
TEXTLIST FX1TextList
  0 = 'Wait For Fixture Home Pos &  Front Door Open'
  10 = 'Wait For Load1 complete & Door Closed'
  20 = 'Wait For Fixture Clamps Closed '
  30 = 'Wait for Trunion move to Pos2'
  40 = 'Wait for Front Door Open for Second load'
  50 = 'Wait for Load2 Complete & Door Closed'
  60 = 'Wait For Fixture Clamps Closed '
  70 = 'Wait For Trunion move to Pos1 '
  80 = 'Wait for Turntable to move Work Pos'
  90 = 'Wait for Weld Start Cmd to R1 & R2 Robot for First Weld'
  100 = 'Wait for Trunion move to Pos2'
  110 = 'Wait for Weld Start Cmd to R1 & R2 Robot for Second Weld'
  120 = 'Wait For Trunion move to Pos1 For Unload '
  130 = 'Wait For Rear Door Open'
  140 = 'Wait for Unload Start Cmd for R3 Robot'
  150 = 'Wait For Fixture Clamps Opened '
  160 = 'Wait for R3 Robot Pick 1 Complete'
  170 = 'Wait for R3 Robot Move to Pounce'
  180 = 'Wait for Trunion move to Pos2'
  190 = 'Wait For Fixture Clamps Opened '
  200 = 'Wait for R3 Robot Pick 2 Complete'
  210 = 'Wait for Trunion move to Pos1'
  220 = 'Wait For Rear Door Closed'
  230 = 'Wait for R3 Robot Drop 1 Complete'
  240 = 'Wait for R3 Robot Drop 2 Complete'
  250 = 'Wait for Tuntable Rotate to Load Position'
   = ''
END_TEXTLIST

// ---- VISUs/Fixture_Auto.TcVIS
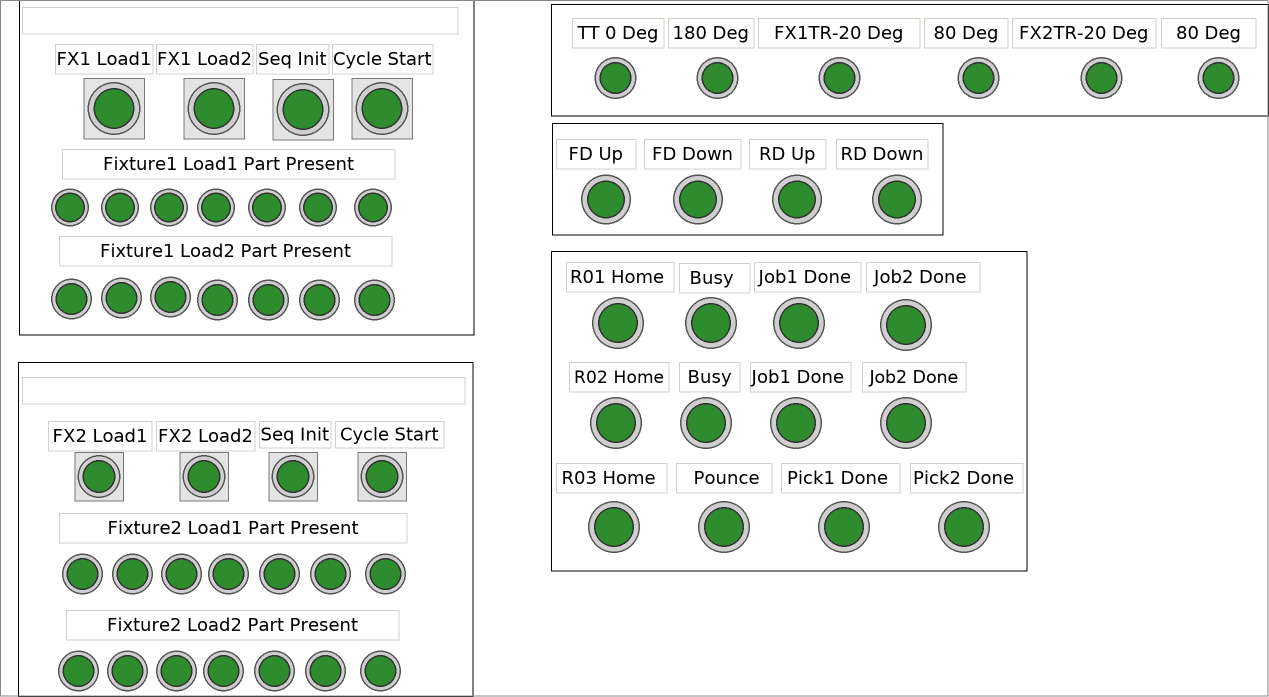
VISUALIZATION Fixture_Auto  // 1269x697
    Rectangle (18,362 455x335)
    Rectangle (19,0 455x335)
    Rectangle (551,4 718x112)
    Rectangle (552,123 391x112)
    Rectangle (551,251 476x320)
    Textfield (55,44 98x30), "FX1 Load1"
    Textfield (156,44 97x30), "FX1 Load2"
    PushSwitch (73,78 82x61), variable: Memory_DB.M_FX1_Load1, behaviour: TAP, style: Switch-PushSwitch-Green
    PushSwitch (173,78 82x61), variable: Memory_DB.M_FX1_Load2, behaviour: TAP, style: Switch-PushSwitch-Green
    Lamp1 (586,54 59x48), variable: Memory_DB.M_Turntable_POS1_Reached, style: Lamp-Lamp1-Green
    Textfield (572,18 92x30), "TT 0 Deg"
    Lamp1 (688,54 59x48), variable: Memory_DB.M_Turntable_POS2_Reached, style: Lamp-Lamp1-Green
    Textfield (668,18 86x30), "180 Deg"
    Textfield (256,44 73x30), "Seq Init"
    PushSwitch (262,79 82x61), variable: Memory_DB.M_FX1_All_Initialise, behaviour: TAP, style: Switch-PushSwitch-Green
    Lamp1 (810,54 59x48), variable: Memory_DB.M_Fixture1_TR_POS1_Reached, style: Lamp-Lamp1-Green
    Textfield (758,18 162x30), "FX1TR-20 Deg"
    Lamp1 (949,54 59x48), variable: Memory_DB.M_Fixture1_TR_POS2_Reached, style: Lamp-Lamp1-Green
    Textfield (924,18 84x30), "80 Deg"
    Lamp1 (571,171 70x57), variable: Inputs.i_Front_Door_Up, style: Lamp-Lamp1-Green
    Textfield (556,139 80x30), "FD Up"
    Lamp1 (663,171 70x57), variable: Inputs.i_Front_Door_Down, style: Lamp-Lamp1-Green
    Textfield (644,139 97x30), "FD Down"
    Lamp1 (762,171 70x57), variable: Inputs.i_Rear_Door_Up, style: Lamp-Lamp1-Green
    Textfield (749,139 77x30), "RD Up"
    Lamp1 (862,171 70x57), variable: Inputs.i_Rear_Door_Down, style: Lamp-Lamp1-Green
    Textfield (836,139 92x30), "RD Down"
    Lamp1 (588,293 60x60), variable: Memory_DB.M_R01_Home, style: Lamp-Lamp1-Green
    Textfield (566,262 108x30), "R01 Home"
    Lamp1 (769,293 60x60), variable: Memory_DB.M_R01_Job_Done1, style: Lamp-Lamp1-Green
    Textfield (754,262 107x30), "Job1 Done"
    Lamp1 (586,393 60x60), variable: Memory_DB.M_R02_Home, style: Lamp-Lamp1-Green
    Textfield (569,362 100x30), "R02 Home"
    Lamp1 (766,393 60x60), variable: Memory_DB.M_R02_Job_Done1, style: Lamp-Lamp1-Green
    Textfield (750,362 101x30), "Job1 Done"
    Lamp1 (579,497 70x60), variable: Memory_DB.M_R03_MH_AtHome, style: Lamp-Lamp1-Green
    Textfield (556,463 111x30), "R03 Home"
    Lamp1 (689,497 70x60), variable: Memory_DB.M_R03_MH_AtPounce, style: Lamp-Lamp1-Green
    Textfield (676,463 96x30), "Pounce"
    Lamp1 (929,497 70x60), variable: Memory_DB.M_R03_MH_Pick2_Done, style: Lamp-Lamp1-Green
    Textfield (910,463 113x30), "Pick2 Done"
    Lamp1 (809,497 70x60), variable: Memory_DB.M_R03_MH_Pick1_Done, style: Lamp-Lamp1-Green
    Textfield (781,463 119x30), "Pick1 Done"
    Lamp1 (48,184 44x47), variable: Inputs.i_FX1_PART_CONTROL_B1, style: Lamp-Lamp1-Green
    Textfield (62,149 333x30), "Fixture1 Load1 Part Present"
    Lamp1 (98,184 44x47), variable: Inputs.i_FX1_PART_CONTROL_B2, style: Lamp-Lamp1-Green
    Lamp1 (147,184 44x47), variable: Inputs.i_FX1_PART_CONTROL_B3, style: Lamp-Lamp1-Green
    Lamp1 (194,184 44x47), variable: Inputs.i_FX1_PART_CONTROL_B4, style: Lamp-Lamp1-Green
    Lamp1 (245,184 44x47), variable: Inputs.i_FX1_PART_CONTROL_B5, style: Lamp-Lamp1-Green
    Lamp1 (296,184 44x47), variable: Inputs.i_FX1_PART_CONTROL_B6, style: Lamp-Lamp1-Green
    Lamp1 (351,184 44x47), variable: Inputs.i_FX1_PART_CONTROL_B7, style: Lamp-Lamp1-Green
    Lamp1 (48,273 47x52), variable: Inputs.i_FX1_PART_CONTROL_B15, style: Lamp-Lamp1-Green
    Textfield (59,236 333x30), "Fixture1 Load2 Part Present"
    Lamp1 (98,272 47x52), variable: Inputs.i_FX1_PART_CONTROL_B16, style: Lamp-Lamp1-Green
    Lamp1 (147,271 47x52), variable: Inputs.i_FX1_PART_CONTROL_B17, style: Lamp-Lamp1-Green
    Lamp1 (194,274 47x52), variable: Inputs.i_FX1_PART_CONTROL_B18, style: Lamp-Lamp1-Green
    Lamp1 (245,274 47x52), variable: Inputs.i_FX1_PART_CONTROL_B19, style: Lamp-Lamp1-Green
    Lamp1 (296,274 47x52), variable: Inputs.i_FX1_PART_CONTROL_B20, style: Lamp-Lamp1-Green
    Lamp1 (351,274 47x52), variable: Inputs.i_FX1_PART_CONTROL_B21, style: Lamp-Lamp1-Green
    Lamp1 (876,295 60x60), variable: Memory_DB.M_R01_Job_Done2, style: Lamp-Lamp1-Green
    Textfield (866,262 114x30), "Job2 Done"
    Lamp1 (876,393 60x60), variable: Memory_DB.M_R02_Job_Done2, style: Lamp-Lamp1-Green
    Textfield (862,362 104x30), "Job2 Done"
    Lamp1 (676,393 60x60), variable: Memory_DB.M_R02_Busy, style: Lamp-Lamp1-Green
    Lamp1 (681,293 60x60), variable: Memory_DB.M_R01_Busy, style: Lamp-Lamp1-Green
    Textfield (679,263 71x30), "Busy"
    Textfield (679,362 61x30), "Busy"
    Textfield (332,44 101x30), "Cycle Start"
    PushSwitch (341,78 82x61), variable: Memory_DB.M_FX1_Cycle_Start_PB, behaviour: TAP, style: Switch-PushSwitch-Green
    Textfield (48,421 104x30), "FX2 Load1"
    Textfield (156,421 99x30), "FX2 Load2"
    PushSwitch (67,452 64x49), variable: Memory_DB.M_FX2_Load1, behaviour: TAP, style: Switch-PushSwitch-Green
    PushSwitch (172,452 64x49), variable: Memory_DB.M_FX2_Load2, behaviour: TAP, style: Switch-PushSwitch-Green
    Textfield (259,421 72x27), "Seq Init"
    PushSwitch (261,452 64x49), variable: Memory_DB.M_FX2_All_Initialise, behaviour: TAP, style: Switch-PushSwitch-Green
    Lamp1 (59,548 47x52), variable: Inputs.i_FX2_PART_CONTROL_B1, style: Lamp-Lamp1-Green
    Textfield (59,513 348x30), "Fixture2 Load1 Part Present"
    Lamp1 (109,548 47x52), variable: Inputs.i_FX2_PART_CONTROL_B2, style: Lamp-Lamp1-Green
    Lamp1 (158,548 47x52), variable: Inputs.i_FX2_PART_CONTROL_B3, style: Lamp-Lamp1-Green
    Lamp1 (205,548 47x52), variable: Inputs.i_FX2_PART_CONTROL_B4, style: Lamp-Lamp1-Green
    Lamp1 (256,548 47x52), variable: Inputs.i_FX2_PART_CONTROL_B5, style: Lamp-Lamp1-Green
    Lamp1 (307,548 47x52), variable: Inputs.i_FX2_PART_CONTROL_B6, style: Lamp-Lamp1-Green
    Lamp1 (362,548 47x52), variable: Inputs.i_FX2_PART_CONTROL_B7, style: Lamp-Lamp1-Green
    Lamp1 (55,645 47x52), variable: Inputs.i_FX2_PART_CONTROL_B15, style: Lamp-Lamp1-Green
    Textfield (66,610 333x30), "Fixture2 Load2 Part Present"
    Lamp1 (104,645 47x52), variable: Inputs.i_FX2_PART_CONTROL_B16, style: Lamp-Lamp1-Green
    Lamp1 (153,645 47x52), variable: Inputs.i_FX2_PART_CONTROL_B17, style: Lamp-Lamp1-Green
    Lamp1 (200,645 47x52), variable: Inputs.i_FX2_PART_CONTROL_B18, style: Lamp-Lamp1-Green
    Lamp1 (251,645 47x52), variable: Inputs.i_FX2_PART_CONTROL_B19, style: Lamp-Lamp1-Green
    Lamp1 (302,645 47x52), variable: Inputs.i_FX2_PART_CONTROL_B20, style: Lamp-Lamp1-Green
    Lamp1 (357,645 47x52), variable: Inputs.i_FX2_PART_CONTROL_B21, style: Lamp-Lamp1-Green
    Lamp1 (1072,54 59x48), variable: Memory_DB.M_Fixture2_TR_POS1_Reached, style: Lamp-Lamp1-Green
    Textfield (1012,18 144x30), "FX2TR-20 Deg"
    Lamp1 (1189,54 59x48), variable: Memory_DB.M_Fixture2_TR_POS2_Reached, style: Lamp-Lamp1-Green
    Textfield (1161,18 95x30), "80 Deg"
    PushSwitch (350,452 64x49), variable: Memory_DB.M_FX2_Cycle_Start_PB, behaviour: TAP, style: Switch-PushSwitch-Green
    Textfield (335,421 109x27), "Cycle Start"
    Textfield (22,7 436x27), text list: 'FX1TextList', text index: Fixture1_Auto.nState_Door
    Textfield (22,377 443x27), text list: 'FX2TextList', text index: Fixture2_Auto.nState_Door
END_VISUALIZATION

// ---- VISUs/Fixture_Manual.TcVIS
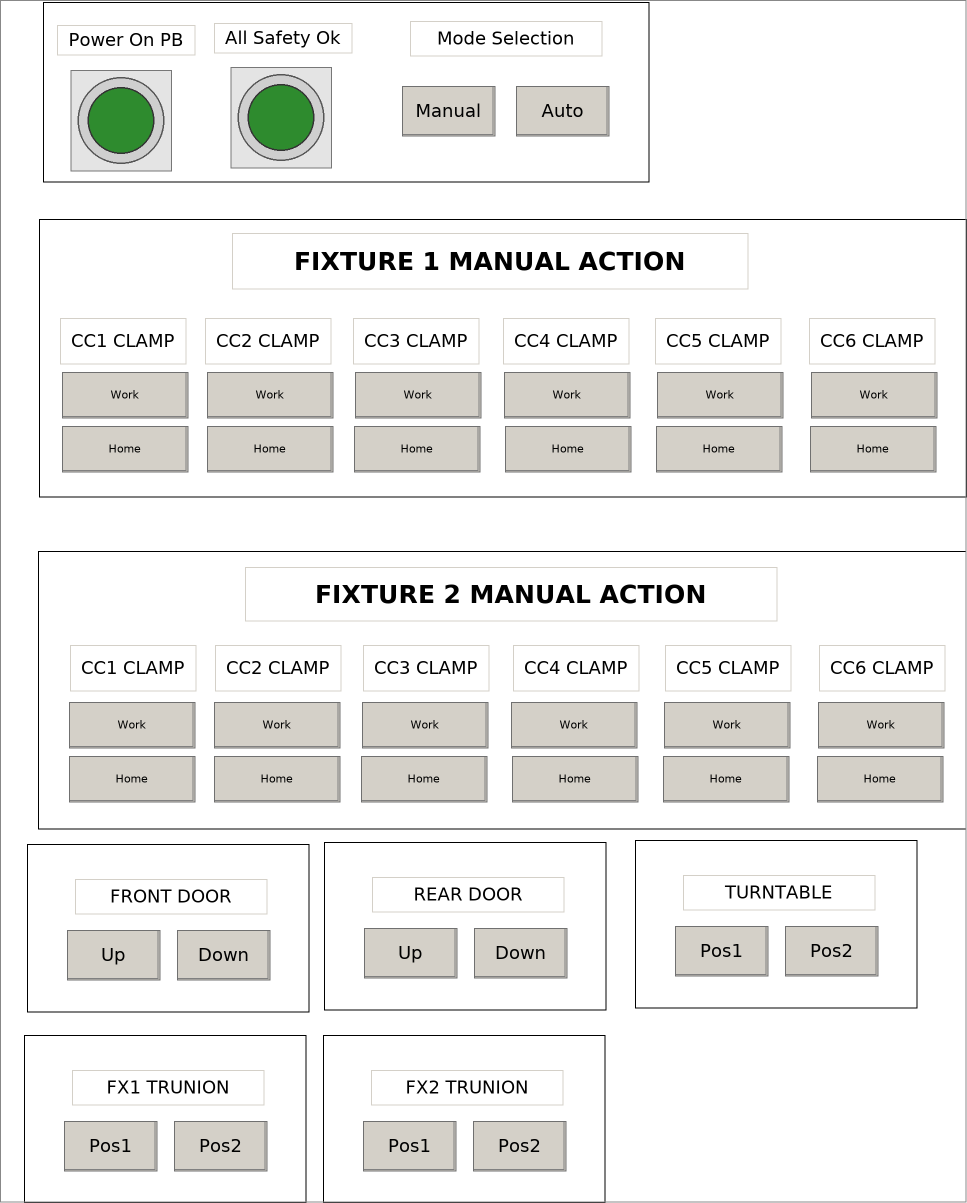
VISUALIZATION Fixture_Manual  // 967x1203
    Rectangle (27,844 282x168)
    Rectangle (38,551 928x278)
    Rectangle (39,219 928x278)
    Rectangle (43,2 606x180)
    Textfield (232,233 516x56), "FIXTURE 1 MANUAL ACTION"
    Button (62,372 126x46), "Work", colour toggle: Inputs.i_FX1_CC1_Clamp_1_Sensor_WP
        tap Memory_DB.M_FX1_CC1_CLAMPING_UNIT1_3_WP
    Button (62,426 126x46), "Home", colour toggle: Inputs.i_FX1_CC1_Clamp_1_Sensor_HP
        tap Memory_DB.M_FX1_CC1_CLAMPING_UNIT1_3_HP
    Textfield (60,318 126x46), "CC1 CLAMP"
    Button (355,372 126x46), "Work", colour toggle: Inputs.i_FX1_CC3_Clamp_1_Sensor_WP
        tap Memory_DB.M_FX1_CC3_CLAMPING_UNIT3_3_WP
    Button (354,426 126x46), "Home", colour toggle: Inputs.i_FX1_CC3_Clamp_1_Sensor_HP
        tap Memory_DB.M_FX1_CC3_CLAMPING_UNIT3_3_HP
    Button (504,372 126x46), "Work", colour toggle: Inputs.i_FX1_CC4_Clamp_1_Sensor_WP
        tap Memory_DB.M_FX1_CC4_CLAMPING_UNIT4_3_WP
    Button (505,426 126x46), "Home", colour toggle: Inputs.i_FX1_CC4_Clamp_1_Sensor_HP
        tap Memory_DB.M_FX1_CC4_CLAMPING_UNIT4_3_HP
    Button (657,372 126x46), "Work", colour toggle: Inputs.i_FX1_CC5_Clamp_1_Sensor_WP
        tap Memory_DB.M_FX1_CC5_CLAMPING_UNIT5_1_WP
    Button (656,426 126x46), "Home", colour toggle: Inputs.i_FX1_CC5_Clamp_1_Sensor_HP
        tap Memory_DB.M_FX1_CC5_CLAMPING_UNIT5_1_HP
    Button (811,372 126x46), "Work", colour toggle: Inputs.i_FX1_CC6_Clamp_1_Sensor_WP
        tap Memory_DB.M_FX1_CC6_CLAMPING_UNIT6_1_WP
    Button (810,426 126x46), "Home", colour toggle: Inputs.i_FX1_CC6_Clamp_1_Sensor_HP
        tap Memory_DB.M_FX1_CC6_CLAMPING_UNIT6_1_hP
    Button (207,372 126x46), "Work", colour toggle: Inputs.i_FX1_CC2_Clamp_1_Sensor_WP
        tap Memory_DB.M_FX1_CC2_CLAMPING_UNIT2_3_WP
    Button (207,426 126x46), "Home", colour toggle: Inputs.i_FX1_CC2_Clamp_1_Sensor_HP
        tap Memory_DB.M_FX1_CC2_CLAMPING_UNIT2_3_HP
    Textfield (503,318 126x46), "CC4 CLAMP"
    Textfield (655,318 126x46), "CC5 CLAMP"
    Textfield (809,318 126x46), "CC6 CLAMP"
    Textfield (205,318 126x46), "CC2 CLAMP"
    Textfield (353,318 126x46), "CC3 CLAMP"
    Textfield (245,567 532x54), "FIXTURE 2 MANUAL ACTION"
    Textfield (70,645 126x46), "CC1 CLAMP"
    Textfield (513,645 126x46), "CC4 CLAMP"
    Textfield (665,645 126x46), "CC5 CLAMP"
    Textfield (819,645 126x46), "CC6 CLAMP"
    Textfield (215,645 126x46), "CC2 CLAMP"
    Textfield (363,645 126x46), "CC3 CLAMP"
    PushSwitch (66,70 110x101), variable: Inputs.i_Power_On_PB, behaviour: TOGGLE, style: Switch-PushSwitch-Green
    Textfield (57,25 138x30), "Power On PB"
    PushSwitch (226,67 110x101), variable: Memory_DB.M_Safety_Ok, behaviour: TOGGLE, style: Switch-PushSwitch-Green
    Textfield (214,23 138x30), "All Safety Ok"
    Button (402,86 93x50), "Manual", text variable: Inputs.i_Mode_Select, colour toggle: Memory_DB.M_Manual_Active
        OnMouseClick: write the text variable via VisuDialogs.Numpad
    Textfield (410,21 192x35), "Mode Selection"
    Button (516,86 93x50), "Auto", text variable: Inputs.i_Mode_Select, colour toggle: Memory_DB.M_Auto_Active
        OnMouseClick: write the text variable via VisuDialogs.Numpad
    Button (69,702 126x46), "Work", colour toggle: Inputs.i_FX2_CC1_Clamp_1_Sensor_WP
        tap Memory_DB.M_FX2_CC1_CLAMPING_UNIT1_3_WP
    Button (69,756 126x46), "Home", colour toggle: Inputs.i_FX2_CC1_Clamp_1_Sensor_HP
        tap Memory_DB.M_FX2_CC1_CLAMPING_UNIT1_3_HP
    Button (362,702 126x46), "Work", colour toggle: Inputs.i_FX2_CC3_Clamp_1_Sensor_WP
        tap Memory_DB.M_FX2_CC3_CLAMPING_UNIT3_3_WP
    Button (361,756 126x46), "Home", colour toggle: Inputs.i_FX2_CC3_Clamp_1_Sensor_HP
        tap Memory_DB.M_FX2_CC3_CLAMPING_UNIT3_3_HP
    Button (511,702 126x46), "Work", colour toggle: Inputs.i_FX2_CC4_Clamp_1_Sensor_WP
        tap Memory_DB.M_FX2_CC4_CLAMPING_UNIT4_3_WP
    Button (512,756 126x46), "Home", colour toggle: Inputs.i_FX2_CC4_Clamp_1_Sensor_HP
        tap Memory_DB.M_FX2_CC4_CLAMPING_UNIT4_3_HP
    Button (664,702 126x46), "Work", colour toggle: Inputs.i_FX2_CC5_Clamp_1_Sensor_WP
        tap Memory_DB.M_FX2_CC5_CLAMPING_UNIT5_1_WP
    Button (663,756 126x46), "Home", colour toggle: Inputs.i_FX2_CC5_Clamp_1_Sensor_HP
        tap Memory_DB.M_FX2_CC5_CLAMPING_UNIT5_1_HP
    Button (818,702 126x46), "Work", colour toggle: Inputs.i_FX2_CC6_Clamp_1_Sensor_WP
        tap Memory_DB.M_FX2_CC6_CLAMPING_UNIT6_1_WP
    Button (817,756 126x46), "Home", colour toggle: Inputs.i_FX2_CC6_Clamp_1_Sensor_HP
        tap Memory_DB.M_FX2_CC6_CLAMPING_UNIT6_1_hP
    Button (214,702 126x46), "Work", colour toggle: Inputs.i_FX2_CC2_Clamp_1_Sensor_WP
        tap Memory_DB.M_FX2_CC2_CLAMPING_UNIT2_3_WP
    Button (214,756 126x46), "Home", colour toggle: Inputs.i_FX2_CC2_Clamp_1_Sensor_HP
        tap Memory_DB.M_FX2_CC2_CLAMPING_UNIT2_3_HP
    Textfield (75,879 192x35), "FRONT DOOR"
    Button (67,930 93x50), "Up", text variable: Inputs.i_Mode_Select, colour toggle: Inputs.i_Front_Door_Up
        tap Memory_DB.M_FRONT_DOOR_UP
    Button (177,930 93x50), "Down", text variable: Inputs.i_Mode_Select, colour toggle: Inputs.i_Front_Door_Down
        tap Memory_DB.M_FRONT_DOOR_DOWN
    Rectangle (324,842 282x168)
    Textfield (372,877 192x35), "REAR DOOR"
    Button (364,928 93x50), "Up", text variable: Inputs.i_Mode_Select, colour toggle: Inputs.i_Rear_Door_Up
        tap Memory_DB.M_REAR_DOOR_UP
    Button (474,928 93x50), "Down", text variable: Inputs.i_Mode_Select, colour toggle: Inputs.i_Rear_Door_Down
        tap Memory_DB.M_REAR_DOOR_DOWN
    Rectangle (635,840 282x168)
    Textfield (683,875 192x35), "TURNTABLE"
    Button (675,926 93x50), "Pos1", text variable: Inputs.i_Mode_Select, colour toggle: Memory_DB.M_Turntable_POS1_Reached
        tap Memory_DB.M_Turntable_POS1_CMD
    Button (785,926 93x50), "Pos2", text variable: Inputs.i_Mode_Select, colour toggle: Memory_DB.M_Turntable_POS2_Reached
        tap Memory_DB.M_Turntable_POS2_CMD
    Rectangle (24,1035 282x168)
    Textfield (72,1070 192x35), "FX1 TRUNION"
    Button (64,1121 93x50), "Pos1", text variable: Inputs.i_Mode_Select, colour toggle: Memory_DB.M_Fixture1_TR_POS1_Reached
        tap Memory_DB.M_Fixture1_TR_POS1_CMD
    Button (174,1121 93x50), "Pos2", text variable: Inputs.i_Mode_Select, colour toggle: Memory_DB.M_Fixture1_TR_POS2_Reached
        tap Memory_DB.M_Fixture1_TR_POS2_CMD
    Rectangle (323,1035 282x168)
    Textfield (371,1070 192x35), "FX2 TRUNION"
    Button (363,1121 93x50), "Pos1", text variable: Inputs.i_Mode_Select, colour toggle: Memory_DB.M_Fixture2_TR_POS1_Reached
        tap Memory_DB.M_Fixture2_TR_POS1_CMD
    Button (473,1121 93x50), "Pos2", text variable: Inputs.i_Mode_Select, colour toggle: Memory_DB.M_Fixture2_TR_POS2_Reached
        tap Memory_DB.M_Fixture2_TR_POS2_CMD
END_VISUALIZATION
